// TwinCAT 3 PLC project ShutterMotion
// ProgramVersion: 3.1.4020.4
// libraries:
//   Tc2_Drive, * (Beckhoff Automation GmbH)
//   Tc2_EtherCAT, * (Beckhoff Automation GmbH)
//   Tc2_MC2, * (Beckhoff Automation GmbH)
//   Tc2_MC2_Drive, * (Beckhoff Automation GmbH)
//   Tc2_NcDrive, * (Beckhoff Automation GmbH)
//   Tc2_Standard, * (Beckhoff Automation GmbH)
//   Tc2_System, * (Beckhoff Automation GmbH)
//   Tc2_Utilities, * (Beckhoff Automation GmbH)
//   Tc3_MC2_AdvancedHoming, * (Beckhoff Automation GmbH)
//   Tc3_Module, * (Beckhoff Automation GmbH)
//   Util, * (System)
//   VisuDialogs, * (System)
// project tree:
//   DUTs/AxisStruct/ ST_AxisGroup.TcDUT, ST_Hall.TcDUT, ST_Track.TcDUT
//   DUTs/CCSInterface STRUCT/CCS to PLC/ ST_Calibrate.TcDUT, ST_ChangeAxisEnable.TcDUT, ST_ChangeBrakeState.TcDUT, ST_ClearAllFaults.TcDUT, ST_ClearAxisFaults.TcDUT, ST_CloseShutter.TcDUT, ST_DisableAllAxes.TcDUT, ST_EnableAllAxes.TcDUT, ST_GoToProd.TcDUT, ST_HomeAxis.TcDUT, ST_MoveAxisAbsolute.TcDUT, ST_MoveAxisRelative.TcDUT, ST_OpenShutter.TcDUT, ST_Reset.TcDUT, ST_TakeExposure.TcDUT, ST_ToggleSafetyCheck.TcDUT
//   DUTs/CCSInterface STRUCT/PLC to CCS/ AxisStatus.TcDUT, ST_CalibDone.TcDUT, ST_Disable.TcDUT, ST_Enable.TcDUT, ST_EncoderSample.TcDUT, ST_Error.TcDUT, ST_HallTransition.TcDUT, ST_Ignored.TcDUT, ST_MotionDone.TcDUT, ST_ShutterStatus.TcDUT, ST_Timer.TcDUT
//   DUTs/CCSInterface STRUCT/ ST_MsgToCCS.TcDUT, ST_MsgToPLC.TcDUT, ST_PLCMsg.TcDUT
//   DUTs/ENUM/ E_Commands.TcDUT, E_Components.TcDUT
//   DUTs/ENUM/State ENUM/ E_StatesEnabled.TcDUT, E_StatesMaint.TcDUT, E_StatesProd.TcDUT, E_StatesTop.TcDUT
//   DUTs/ ST_PtpDiag.TcDUT, T_MioSysTimes.TcDUT, T_TaskStartTimes.TcDUT
//   / GlobalTextList.TcGTLO, PlcTaskMain.TcTTO, Visualization Manager.TcVMO (not stored)
//   GVLs/ GVL.TcGVL
//   POUs/ FB_Power.TcPOU, FB_Protection.TcPOU, FB_PtpDiagReader.TcPOU, F_MioExtTime.TcPOU, F_HaveDifferentIDs.TcPOU, MAIN.TcPOU
//   POUs/StateMachine/ FB_Cycler.TcPOU, FB_ShutterSM.TcPOU, FB_Tracking.TcPOU
//   POUs/StateMachine/StateTop/ FB_StateDisabled.TcPOU, FB_StateEnabled.TcPOU
//   POUs/StateMachine/StateTop/StateEnabled/ FB_Reset.TcPOU, FB_StateMaint.TcPOU, FB_StateProd.TcPOU
//   POUs/StateMachine/StateTop/StateEnabled/StateMaint/ FB_Homing.TcPOU, FB_StateCalibrating.TcPOU, FB_StateMoving.TcPOU, FB_StateStill.TcPOU
//   POUs/StateMachine/StateTop/StateEnabled/StateProd/ FB_StateClosed.TcPOU, FB_StateClosing.TcPOU, FB_StateOpened.TcPOU, FB_StateOpening.TcPOU, FB_StateTravelling.TcPOU
//   VISUs/ Visualization.TcVIS
// real-time tasks:
//   TASK PlcTaskMain: cycle T#500us, priority 20, ADS port 350
// motion (NC):
//   TASK NC-Task 1 SAF: cycle T#500us, priority 1, ADS port 501
//   TASK NC-Task 1 SVB: cycle T#5ms, priority 40, ADS port 511
//   AXIS XP (id 1)
//     Dynamic: Acceleration=7407.41, Deceleration=7407.41, Jerk=32921.8
//     Velo: RefSearch=60, SlowManual=150
//     OtherSettings: AllowMotionCmdToSlave=true
//     encoder EncType=4
//       EncPara: ScaleFactorNumerator=0.0498327596, MaxCount=#x0000ffff
//         SoftEndMaxControl: Range=749
//         Inc: RefSearchInverse=true, RefSyncInverse=false, RefSoftSyncMask=#x0000ffff
//         TimeComp: TimeCompMode=1, EncDelayCycles=4
//     drive DrvType=24
//       Analog: VeloReferenz=2038.894
//       TimeComp: TaskDelayCycles=1
//     controller CtrType=1
//       CtrPara: PriorControlFactor=1
//         PosDiffControl: Range=2.5, Time=0.01
//         Observer: BandWidth=20
//   AXIS XM (id 2)
//     Dynamic: Acceleration=7407.41, Deceleration=7407.41, Jerk=32921.8
//     Velo: RefSearch=60
//     OtherSettings: AllowMotionCmdToSlave=true
//     encoder EncType=4
//       EncPara: ScaleFactorNumerator=0.0498327596, MaxCount=#x0000ffff
//         SoftEndMaxControl: Range=749
//         Inc: RefSoftSyncMask=#x0000ffff
//         TimeComp: TimeCompMode=1, EncDelayCycles=4
//     drive DrvType=24
//       Analog: VeloReferenz=2038.894
//       TimeComp: TaskDelayCycles=1
//     controller CtrType=1
//       CtrPara: PriorControlFactor=1
//         PosDiffControl: Range=2.5, Time=0.01
//         Observer: BandWidth=20
// I/O:
//   DEVICE Device 1 (EtherCAT), AmsNetId 10.0.1.28.2.1
//     MCD-00 (EK1200) [EK1200-5000 EtherCAT Power supply (2A E-Bus)]
//       MBC-00 (EL9570) [EL9570 Buffer capacitor terminal]
//       MDR-00 (EL7047) [EL7047 1Ch. Stepper motor output stage (50V, 5A)]
//       MPD-00 (EL9184) [EL9184 Potential Connection, 8 x 24V, 8 x Ground]
//       MIO-00 (EL1259) [EL1259 8Ch. Dig Input 24V/8Ch. Dig. Output 24V with Multi-Time-Stamp]
//       MIO-01 (EL1259) [EL1259 8Ch. Dig Input 24V/8Ch. Dig. Output 24V with Multi-Time-Stamp]
//       MTC-00 (EL3214) [EL3214 4Ch. Ana. Input PT100 (RTD)]
//       MBC-01 (EL9570) [EL9570 Buffer capacitor terminal]
//       MDR-01 (EL7047) [EL7047 1Ch. Stepper motor output stage (50V, 5A)]
//       MRE-01 (EL2622) [EL2622 2Ch. Relay Output, NO (230V AC / 30V DC)]
//       MTM-00 (EL6688) [EL6688 - External Synchronisation Interface (IEEE1588)]
//       END (EL9011) [EL9011 End Terminal]
// variable links:
//   (this object) <-> Device 1 (EtherCAT)/MCD-00 (EK1200)/MDR-00 (EL7047)
//     Drive/Inputs/In/nState1 @bit 3 <-> STM Status/Status/Error
//     Drive/Inputs/In/nState1 @bit 7 <-> STM Status/Status/Motor stall
//     Drive/Inputs/In/nState1 @bit 5 <-> STM Status/Status/Moving negative
//     Drive/Inputs/In/nState1 @bit 4 <-> STM Status/Status/Moving positive
//     Drive/Inputs/In/nState1 @bit 1 <-> STM Status/Status/Ready
//     Drive/Inputs/In/nState1 <-> STM Status/Status/Ready to enable
//     Drive/Inputs/In/nState1 @bit 6 <-> STM Status/Status/Torque reduced
//     Drive/Inputs/In/nState1 @bit 2 <-> STM Status/Status/Warning
//     Drive/Inputs/In/nState2 @bit 5 <-> STM Status/Status/Sync error
//     Drive/Inputs/In/nState2 @bit 7 <-> STM Status/Status/TxPDO Toggle
//     Drive/Inputs/In/nState4 @bit 1 <-> WcState/InputToggle
//     Drive/Outputs/Out/nCtrl1 <-> STM Control/Control/Enable
//     Drive/Outputs/Out/nCtrl1 @bit 2 <-> STM Control/Control/Reduce torque
//     Drive/Outputs/Out/nCtrl1 @bit 1 <-> STM Control/Control/Reset
//     Drive/Outputs/Out/nCtrl2 @bit 3 <-> STM Control/Control/Digital output 1
//     Drive/Outputs/Out/nDataOut2[0] <-> STM Velocity/Velocity
//     Enc/Inputs/In/nDataIn1[0] <-> ENC Status compact/Counter value
//     Enc/Inputs/In/nDataIn2[0] <-> ENC Status compact/Latch value
//     Enc/Inputs/In/nState1 @bit 4 <-> ENC Status compact/Status/Counter overflow
//     Enc/Inputs/In/nState1 @bit 3 <-> ENC Status compact/Status/Counter underflow
//     Enc/Inputs/In/nState1 @bit 7 <-> ENC Status compact/Status/Extrapolation stall
//     Enc/Inputs/In/nState1 <-> ENC Status compact/Status/Latch C valid
//     Enc/Inputs/In/nState1 @bit 1 <-> ENC Status compact/Status/Latch extern valid
//     Enc/Inputs/In/nState1 @bit 2 <-> ENC Status compact/Status/Set counter done
//     Enc/Inputs/In/nState2 @bit 4 <-> ENC Status compact/Status/Status of extern latch
//     Enc/Inputs/In/nState2 <-> ENC Status compact/Status/Status of input A
//     Enc/Inputs/In/nState2 @bit 1 <-> ENC Status compact/Status/Status of input B
//     Enc/Inputs/In/nState2 @bit 2 <-> ENC Status compact/Status/Status of input C
//     Enc/Inputs/In/nState2 @bit 5 <-> ENC Status compact/Status/Sync error
//     Enc/Inputs/In/nState2 @bit 7 <-> ENC Status compact/Status/TxPDO Toggle
//     Enc/Inputs/In/nState4 @bit 1 <-> WcState/InputToggle
//     Enc/Outputs/Out/nCtrl1 <-> ENC Control compact/Control/Enable latch C
//     Enc/Outputs/Out/nCtrl1 @bit 3 <-> ENC Control compact/Control/Enable latch extern on negative edge
//     Enc/Outputs/Out/nCtrl1 @bit 1 <-> ENC Control compact/Control/Enable latch extern on positive edge
//     Enc/Outputs/Out/nCtrl1 @bit 2 <-> ENC Control compact/Control/Set counter
//     Enc/Outputs/Out/nDataOut1[0] <-> ENC Control compact/Set counter value
//   (this object) <-> Device 1 (EtherCAT)/MCD-00 (EK1200)/MDR-01 (EL7047)
//     Drive/Inputs/In/nState1 @bit 3 <-> STM Status/Status/Error
//     Drive/Inputs/In/nState1 @bit 7 <-> STM Status/Status/Motor stall
//     Drive/Inputs/In/nState1 @bit 5 <-> STM Status/Status/Moving negative
//     Drive/Inputs/In/nState1 @bit 4 <-> STM Status/Status/Moving positive
//     Drive/Inputs/In/nState1 @bit 1 <-> STM Status/Status/Ready
//     Drive/Inputs/In/nState1 <-> STM Status/Status/Ready to enable
//     Drive/Inputs/In/nState1 @bit 6 <-> STM Status/Status/Torque reduced
//     Drive/Inputs/In/nState1 @bit 2 <-> STM Status/Status/Warning
//     Drive/Inputs/In/nState2 @bit 5 <-> STM Status/Status/Sync error
//     Drive/Inputs/In/nState2 @bit 7 <-> STM Status/Status/TxPDO Toggle
//     Drive/Inputs/In/nState4 @bit 1 <-> WcState/InputToggle
//     Drive/Outputs/Out/nCtrl1 <-> STM Control/Control/Enable
//     Drive/Outputs/Out/nCtrl1 @bit 2 <-> STM Control/Control/Reduce torque
//     Drive/Outputs/Out/nCtrl1 @bit 1 <-> STM Control/Control/Reset
//     Drive/Outputs/Out/nCtrl2 @bit 3 <-> STM Control/Control/Digital output 1
//     Drive/Outputs/Out/nDataOut2[0] <-> STM Velocity/Velocity
//     Enc/Inputs/In/nDataIn1[0] <-> ENC Status compact/Counter value
//     Enc/Inputs/In/nDataIn2[0] <-> ENC Status compact/Latch value
//     Enc/Inputs/In/nState1 @bit 4 <-> ENC Status compact/Status/Counter overflow
//     Enc/Inputs/In/nState1 @bit 3 <-> ENC Status compact/Status/Counter underflow
//     Enc/Inputs/In/nState1 @bit 7 <-> ENC Status compact/Status/Extrapolation stall
//     Enc/Inputs/In/nState1 <-> ENC Status compact/Status/Latch C valid
//     Enc/Inputs/In/nState1 @bit 1 <-> ENC Status compact/Status/Latch extern valid
//     Enc/Inputs/In/nState1 @bit 2 <-> ENC Status compact/Status/Set counter done
//     Enc/Inputs/In/nState2 @bit 4 <-> ENC Status compact/Status/Status of extern latch
//     Enc/Inputs/In/nState2 <-> ENC Status compact/Status/Status of input A
//     Enc/Inputs/In/nState2 @bit 1 <-> ENC Status compact/Status/Status of input B
//     Enc/Inputs/In/nState2 @bit 2 <-> ENC Status compact/Status/Status of input C
//     Enc/Inputs/In/nState2 @bit 5 <-> ENC Status compact/Status/Sync error
//     Enc/Inputs/In/nState2 @bit 7 <-> ENC Status compact/Status/TxPDO Toggle
//     Enc/Inputs/In/nState4 @bit 1 <-> WcState/InputToggle
//     Enc/Outputs/Out/nCtrl1 <-> ENC Control compact/Control/Enable latch C
//     Enc/Outputs/Out/nCtrl1 @bit 3 <-> ENC Control compact/Control/Enable latch extern on negative edge
//     Enc/Outputs/Out/nCtrl1 @bit 1 <-> ENC Control compact/Control/Enable latch extern on positive edge
//     Enc/Outputs/Out/nCtrl1 @bit 2 <-> ENC Control compact/Control/Set counter
//     Enc/Outputs/Out/nDataOut1[0] <-> ENC Control compact/Set counter value
//   ShutterMotion Instance <-> Device 1 (EtherCAT)
//     PlcTaskMain Inputs/GVL.DcToExtTimeOffset <-> InfoData/DcToExtTimeOffset
//     PlcTaskMain Inputs/GVL.DcToTcTimeOffset <-> InfoData/DcToTcTimeOffset
//   ShutterMotion Instance <-> Device 1 (EtherCAT)/MCD-00 (EK1200)/MDR-00 (EL7047)
//     PlcTaskMain Inputs/MAIN.fMotorTemp[0] <-> STM Synchron info data/Info data 1
//     PlcTaskMain Inputs/MAIN.stAxis[0].bLimitDeployed <-> STM Status/Status/Digital input 2
//     PlcTaskMain Inputs/MAIN.stAxis[0].bLimitHome <-> STM Status/Status/Digital input 1
//   ShutterMotion Instance <-> Device 1 (EtherCAT)/MCD-00 (EK1200)/MDR-01 (EL7047)
//     PlcTaskMain Inputs/MAIN.fMotorTemp[1] <-> STM Synchron info data/Info data 1
//     PlcTaskMain Inputs/MAIN.stAxis[1].bLimitDeployed <-> STM Status/Status/Digital input 2
//     PlcTaskMain Inputs/MAIN.stAxis[1].bLimitHome <-> STM Status/Status/Digital input 1
//   ShutterMotion Instance <-> Device 1 (EtherCAT)/MCD-00 (EK1200)/MIO-00 (EL1259)
//     PlcTaskMain Inputs/GVL.bInputEventState[{0..7}] <-> MTI Inputs 2x Channel {1..8}/Input event state 1  (8 links)
//     PlcTaskMain Inputs/GVL.mioSysTime[0] <-> DEV Inputs Device/SysTime
//     PlcTaskMain Inputs/GVL.nInputEventTime[{0..7}] <-> MTI Inputs 2x Channel {1..8}/Input event time 1  (8 links)
//     PlcTaskMain Inputs/GVL.nNumOfInputs[{0..7}] <-> MTI Inputs 2x Channel {1..8}/No of input events  (8 links)
//   ShutterMotion Instance <-> Device 1 (EtherCAT)/MCD-00 (EK1200)/MIO-01 (EL1259)
//     PlcTaskMain Inputs/GVL.bInputEventState[{8..14}] <-> MTI Inputs 2x Channel {1..7}/Input event state 1  (7 links)
//     PlcTaskMain Inputs/GVL.mioSysTime[1] <-> DEV Inputs Device/SysTime
//     PlcTaskMain Inputs/GVL.nInputEventTime[{8..14}] <-> MTI Inputs 2x Channel {1..7}/Input event time 1  (7 links)
//     PlcTaskMain Inputs/GVL.nNumOfInputs[{8..14}] <-> MTI Inputs 2x Channel {1..7}/No of input events  (7 links)
//   ShutterMotion Instance <-> Device 1 (EtherCAT)/MCD-00 (EK1200)/MRE-01 (EL2622)
//     PlcTaskMain Outputs/MAIN.stAxis[0].bBrake <-> Channel 1/Output
//     PlcTaskMain Outputs/MAIN.stAxis[1].bBrake <-> Channel 2/Output
//   ShutterMotion Instance <-> Device 1 (EtherCAT)/MCD-00 (EK1200)/MTC-00 (EL3214)
//     PlcTaskMain Inputs/MAIN.fRtdTemp[0] <-> RTD Inputs Channel 1/Value
//     PlcTaskMain Inputs/MAIN.fRtdTemp[1] <-> RTD Inputs Channel 2/Value
//     PlcTaskMain Inputs/MAIN.fRtdTemp[2] <-> RTD Inputs Channel 3/Value
//   ShutterMotion Instance <-> Device 1 (EtherCAT)/MCD-00 (EK1200)/MTM-00 (EL6688)
//     PlcTaskMain Inputs/GVL.ptpAdsAddr <-> InfoData/AdsAddr
//   ShutterMotion Instance <-> NC-Task 1 SAF/Axes/XM
//     PlcTaskMain Inputs/MAIN.stAxis[1].axisRef.NcToPlc <-> Outputs/ToPlc
//     PlcTaskMain Outputs/MAIN.stAxis[1].axisRef.PlcToNc <-> Inputs/FromPlc
//   ShutterMotion Instance <-> NC-Task 1 SAF/Axes/XP
//     PlcTaskMain Inputs/MAIN.stAxis[0].axisRef.NcToPlc <-> Outputs/ToPlc
//     PlcTaskMain Outputs/MAIN.stAxis[0].axisRef.PlcToNc <-> Inputs/FromPlc

CONFIGURATION ShutterMotion
    RESOURCE PLC ON TwinCAT3
        TASK PlcTaskMain(INTERVAL := T#500us, PRIORITY := 20);
        PROGRAM MAIN WITH PlcTaskMain : MAIN;
    END_RESOURCE
END_CONFIGURATION

// ---- DUTs/AxisStruct/ST_AxisGroup.TcDUT
TYPE ST_AxisGroup :
STRUCT
	//basic built in functions
	mcPower		: MC_Power;
	mcReset		: MC_Reset;
	mcMoveAbs	: MC_MoveAbsolute;
	mcMoveRel	: MC_MoveRelative;
	mcHome		: MC_Home;
	mcStop		: MC_Stop;
	mcJog		: MC_Jog; //required for homing routine
	
	//Status
	bIsCalibrated	: BOOL;
	
	//linkable variables
	axisRef					: AXIS_REF;;
	bBrake AT %Q* 			: BOOL;			(* 1-Brake disengaged, 0-Brake engaged *)
	bLimitHome AT %I*		: BOOL;			(* 1-at limit, 0-not at limit. Should be changed to 0-at limit, 1-not at limit to be SIL-2 compliance. Requires hardware change. *)
	bLimitDeployed AT %I*	: BOOL;			(* 1-at limit, 0-not at limit. Should be changed to 0-at limit, 1-not at limit to be SIL-2 compliance. Requires hardware change. *)

	//used for tracking linear motion using hall sensors
	//fbHallSig_rtrig		: ARRAY [GVL.cHallLower .. GVL.cHallUpper] OF R_TRIG;
	//fbHallSig_ftrig 	: ARRAY [GVL.cHallLower .. GVL.cHallUpper] OF F_TRIG;
	fHallPosCal			: ARRAY [GVL.cDirPos .. GVL.cDirNeg, 0 .. GVL.cTripCount] OF LREAL;
	fHallPosAct			: LREAL;
	nHallTime			: UDINT; //unit in nanosecond
	nTripCount 			: INT;
	//nHallSequence		: ARRAY [GVL.cDirPos .. GVL.cDirNeg, 0 .. GVL.cTripCount] OF WORD;
	stHall				: ARRAY [GVL.cDirPos .. GVL.cDirNeg, 0 .. GVL.cTripCount] OF ST_Hall;
	nSeqToCompare		: WORD;
	fPosDiffAtTrip		: LREAL;
	bTrackedFlag		: BOOL;

END_STRUCT
END_TYPE

// ---- DUTs/AxisStruct/ST_Hall.TcDUT
TYPE ST_Hall :
STRUCT
	nSeq	: WORD;
	bEdge	: BOOL; // 1-rising edge, 0-falling edge
END_STRUCT
END_TYPE

// ---- DUTs/AxisStruct/ST_Track.TcDUT
TYPE ST_Track :
STRUCT
	nSeqToCompare 	: WORD;
	bEdgeToCompare	: BOOL;
	tScanTime		: T_DCTIME64;
	nHallID			: DINT;
END_STRUCT
END_TYPE

// ---- DUTs/CCSInterface STRUCT/CCS to PLC/ST_Calibrate.TcDUT
{attribute 'pack_mode' := '1'}
TYPE ST_Calibrate EXTENDS ST_MsgToPLC:
STRUCT
    (* TBD - calibration parameters. *)
END_STRUCT
END_TYPE

// ---- DUTs/CCSInterface STRUCT/CCS to PLC/ST_ChangeAxisEnable.TcDUT
{attribute 'pack_mode' := '1'}
TYPE ST_ChangeAxisEnable EXTENDS ST_MsgToPLC:
STRUCT
    axisIndex	: DINT;
    enabled		: BOOL;
END_STRUCT
END_TYPE

// ---- DUTs/CCSInterface STRUCT/CCS to PLC/ST_ChangeBrakeState.TcDUT
{attribute 'pack_mode' := '1'}
TYPE ST_ChangeBrakeState EXTENDS ST_MsgToPLC:
STRUCT
	axisIndex	: DINT;
    state		: BOOL; (* TRUE=Disengaged, FALSE=Engaged *)
END_STRUCT
END_TYPE

// ---- DUTs/CCSInterface STRUCT/CCS to PLC/ST_ClearAllFaults.TcDUT
{attribute 'pack_mode' := '1'}
TYPE ST_ClearAllFaults EXTENDS ST_MsgToPLC:
STRUCT
END_STRUCT
END_TYPE

// ---- DUTs/CCSInterface STRUCT/CCS to PLC/ST_ClearAxisFaults.TcDUT
{attribute 'pack_mode' := '1'}
TYPE ST_ClearAxisFaults EXTENDS ST_MsgToPLC :
STRUCT
    axisIndex: DINT;
END_STRUCT
END_TYPE

// ---- DUTs/CCSInterface STRUCT/CCS to PLC/ST_CloseShutter.TcDUT
{attribute 'pack_mode' := '1'}
TYPE ST_CloseShutter EXTENDS ST_MsgToPLC:
STRUCT

END_STRUCT
END_TYPE

// ---- DUTs/CCSInterface STRUCT/CCS to PLC/ST_DisableAllAxes.TcDUT
{attribute 'pack_mode' := '1'}
TYPE ST_DisableAllAxes EXTENDS ST_MsgToPLC:
STRUCT
END_STRUCT
END_TYPE

// ---- DUTs/CCSInterface STRUCT/CCS to PLC/ST_EnableAllAxes.TcDUT
{attribute 'pack_mode' := '1'}
TYPE ST_EnableAllAxes EXTENDS ST_MsgToPLC:
STRUCT
END_STRUCT
END_TYPE

// ---- DUTs/CCSInterface STRUCT/CCS to PLC/ST_GoToProd.TcDUT
{attribute 'pack_mode' := '1'}
TYPE ST_GoToProd EXTENDS ST_MsgToPLC:
STRUCT
END_STRUCT
END_TYPE

// ---- DUTs/CCSInterface STRUCT/CCS to PLC/ST_HomeAxis.TcDUT
{attribute 'pack_mode' := '1'}
TYPE ST_HomeAxis EXTENDS ST_MsgToPLC:
STRUCT
    axisIndex: DINT;
END_STRUCT
END_TYPE

// ---- DUTs/CCSInterface STRUCT/CCS to PLC/ST_MoveAxisAbsolute.TcDUT
{attribute 'pack_mode' := '1'}
TYPE ST_MoveAxisAbsolute EXTENDS ST_MsgToPLC:
STRUCT
    axisIndex	: DINT;
    position	: LREAL;
    speed		: LREAL;
END_STRUCT
END_TYPE

// ---- DUTs/CCSInterface STRUCT/CCS to PLC/ST_MoveAxisRelative.TcDUT
{attribute 'pack_mode' := '1'}
TYPE ST_MoveAxisRelative EXTENDS ST_MsgToPLC:
STRUCT
    axisIndex	: DINT;
    distance	: LREAL;
    moveTime	: TIME;
END_STRUCT
END_TYPE

// ---- DUTs/CCSInterface STRUCT/CCS to PLC/ST_OpenShutter.TcDUT
{attribute 'pack_mode' := '1'}
TYPE ST_OpenShutter EXTENDS ST_MsgToPLC:
STRUCT

END_STRUCT
END_TYPE

// ---- DUTs/CCSInterface STRUCT/CCS to PLC/ST_Reset.TcDUT
{attribute 'pack_mode' := '1'}
TYPE ST_Reset EXTENDS ST_MsgToPLC:
STRUCT
    (* TBD - Shutter config info. *)
	speed 			: LREAL;
END_STRUCT
END_TYPE

// ---- DUTs/CCSInterface STRUCT/CCS to PLC/ST_TakeExposure.TcDUT
{attribute 'pack_mode' := '1'}
TYPE ST_TakeExposure EXTENDS ST_MsgToPLC:
STRUCT
    exposureTime: TIME;
END_STRUCT
END_TYPE

// ---- DUTs/CCSInterface STRUCT/CCS to PLC/ST_ToggleSafetyCheck.TcDUT
{attribute 'pack_mode' := '1'}
TYPE ST_ToggleSafetyCheck EXTENDS ST_MsgToPLC :
STRUCT
END_STRUCT
END_TYPE

// ---- DUTs/CCSInterface STRUCT/PLC to CCS/AxisStatus.TcDUT
{attribute 'pack_mode' := '1'}
(*already a built in struct called ST_AxisStatus so leaving this as AxisStatus instead*)
TYPE AxisStatus:
STRUCT
    actPos		: LREAL;	(* Actual position in mm. *)
    actVel		: LREAL;	(* Actual velocity in mm/sec. *)
    setAcc		: LREAL;	(* Set acceleration in mm/sec^2.*)
	enabled		: BOOL;		(* Is the axis enabled? *)
	brakeSet	: BOOL;		(* Is the brake engaged? *)
    lowLimit	: BOOL;		(* Low limit switch tripped? *)
	highLimit	: BOOL; 	(* High limit switch tripped? *)
	isHomed		: BOOL; 	(* Has the axis been homed? *)
	errorID		: UDINT; 	(* Axis error code. *)
    icTemp	: LREAL; 	    (* Temperature of motor controller IC, Celsius. *)
END_STRUCT
END_TYPE

// ---- DUTs/CCSInterface STRUCT/PLC to CCS/ST_CalibDone.TcDUT
{attribute 'pack_mode' := '1'}
TYPE ST_CalibDone EXTENDS ST_MsgToCCS:
STRUCT
    homePosition		: ARRAY [0..1] OF LREAL;
    deployedPosition	: ARRAY [0..1] OF LREAL;
    (* hallPosCal[a, d, t] is coordinate of
       the (t+1)st transition that occurred
       while moving axis a+1 in direction d.
       d=0 for positive, d=1 for negative.
     *)
    hallPosCal			: ARRAY [0..1, 0..1, 0..239] OF LREAL;
END_STRUCT
END_TYPE

// ---- DUTs/CCSInterface STRUCT/PLC to CCS/ST_Disable.TcDUT
{attribute 'pack_mode' := '1'}
TYPE ST_Disable EXTENDS ST_MsgToCCS:
STRUCT
END_STRUCT
END_TYPE

// ---- DUTs/CCSInterface STRUCT/PLC to CCS/ST_Enable.TcDUT
{attribute 'pack_mode' := '1'}
TYPE ST_Enable EXTENDS ST_MsgToCCS:
STRUCT
END_STRUCT
END_TYPE

// ---- DUTs/CCSInterface STRUCT/PLC to CCS/ST_EncoderSample.TcDUT
{attribute 'pack_mode' := '1'}
TYPE ST_EncoderSample:
STRUCT
    extTime	: T_DCTIME64; (* The time of the sample. Beckhoff TAI-like external time.*)
    pos		: LREAL; (* Axis position in mm. *)
END_STRUCT
END_TYPE

// ---- DUTs/CCSInterface STRUCT/PLC to CCS/ST_Error.TcDUT
{attribute 'pack_mode' := '1'}
TYPE ST_Error EXTENDS ST_MsgToCCS:
STRUCT
	errors	: UDINT;
END_STRUCT
END_TYPE

(*
TYPE E_Error:
(
    MOTION_VETOED 	:= 2#1,				//1,
    BRAKE_SET 		:= 2#10,			//2,
    HALL_DIFF 		:= 2#100,			//4,
    SHORT_EXPOSURE 	:= 2#1000,			//8,
    NOT_HOMED 		:= 2#10000,			//16,
    HOME_LIMIT 		:= 2#100000,		//32,
    DEPLOYED_LIMIT 	:= 2#1000000,		//64,
    UNSAFE_MOVE 	:= 2#10000000,		//128,
    TOO_FAST 		:= 2#100000000,		//256,
    AXIS_DISABLED 	:= 2#1000000000,	//512
) UDINT;
END_TYPE

*)

// ---- DUTs/CCSInterface STRUCT/PLC to CCS/ST_HallTransition.TcDUT
{attribute 'pack_mode' := '1'}
TYPE ST_HallTransition:
STRUCT
    id		: DINT; (* ID no. of sensor. *)
    extTime	: T_DCTIME64; (* The time of the transition, Beckhoff TAI-like external time. *)
    pos		: LREAL; (* Position of transition. *)
    on		: BOOL; (* TRUE for off -> on, else FALSE. *)
END_STRUCT
END_TYPE

// ---- DUTs/CCSInterface STRUCT/PLC to CCS/ST_Ignored.TcDUT
{attribute 'pack_mode' := '1'}
TYPE ST_Ignored EXTENDS ST_MsgToCCS:
STRUCT
    reason: DINT;
END_STRUCT
END_TYPE
 
(* Reasons for ignoring an event:
0: Wrong message-set version.
1: Wrong state.
*)

// ---- DUTs/CCSInterface STRUCT/PLC to CCS/ST_MotionDone.TcDUT
{attribute 'pack_mode' := '1'}
TYPE ST_MotionDone EXTENDS ST_MsgToCCS:
STRUCT
    axisNum		: DINT;						(* Which axis moved. *)
    startTime	: T_DCTIME64;				(* When motion started. Absolute TAI64N-like nanoseconds since Jan 1, 2000.*)
    startPos	: LREAL;					(* Starting position. *)
    targetDur	: LTIME;					(* Expected duration of motion. *)
    targetPos	: LREAL;					(* Desired final position. *)
    endPos		: LREAL;					(* Actual final position. *)
    actualDur	: LTIME;					(* Actual duration. *)
    ntrans		: DINT;						(* No. of Hall transitions. *)
    maxtrans	: DINT := GVL.cTripCount+1;	(* Size  N of trans array. *)
    nsamples	: DINT;						(* No of encoder samples. *)
    maxsamples	: DINT := GVL.cTripCount+1;	(* Size M of samples array. *)
    trans		: ARRAY [0 .. GVL.cTripCount] OF ST_HallTransition;
    samples		: ARRAY	[0 .. GVL.cTripCount] OF ST_EncoderSample;
	ptpState    : DINT;                     (* Encoded PTP slave clock state. *)
											(* 0=NO_OPERATION, 1=INITIALIZING, 2=FAULTY, 3=DISABLED, 4=LISTENING, *)
											(* 5=PRE_MASTER, 6=MASTER, 7=PASSIVE, 8=UNCALIBRATED, 9=SLAVE. *)
	leapSeconds : DINT;                     (* Latest leap second count gotten from PTP. *)
	leapIsValid : BOOL;                     (* Is nonzero if leap second count is valid, else is zero. *)
END_STRUCT
END_TYPE

// ---- DUTs/CCSInterface STRUCT/PLC to CCS/ST_ShutterStatus.TcDUT
{attribute 'pack_mode' := '1'}
TYPE ST_ShutterStatus EXTENDS ST_MsgToCCS:
STRUCT
    motionProfile	: DINT; (* Motion profile index. *)
    isCalibrated	: BOOL;
    smState			: DINT;
    axis			: ARRAY [0..1] OF AxisStatus;
	isSafetyOn		: BOOL;
	temperature 	: ARRAY [0..2] OF DINT;
	when			: T_DCTIME64;               (* When this message was created, TAI nanoseconds since Jan 1, 2000. *)
	ptpState    	: DINT;                     (* Encoded PTP slave clock state. *)
												(* 0=NO_OPERATION, 1=INITIALIZING, 2=FAULTY, 3=DISABLED, 4=LISTENING, *)
												(* 5=PRE_MASTER, 6=MASTER, 7=PASSIVE, 8=UNCALIBRATED, 9=SLAVE. *)
	leapSeconds		: DINT;                     (* Latest leap second count gotten from PTP. *)
	leapIsValid 	: BOOL;                     (* Is nonzero if leap second count is valid, else is zero. *)
END_STRUCT
END_TYPE

// ---- DUTs/CCSInterface STRUCT/PLC to CCS/ST_Timer.TcDUT
{attribute 'pack_mode' := '1'}
TYPE ST_Timer EXTENDS ST_MsgToCCS:
STRUCT
END_STRUCT
END_TYPE

// ---- DUTs/CCSInterface STRUCT/ST_MsgToCCS.TcDUT
{attribute 'pack_mode' := '1'}
TYPE ST_MsgToCCS EXTENDS ST_PLCMsg:
STRUCT
	sequence: DINT;(* Increment this to ensure notification. *)
END_STRUCT
END_TYPE

// ---- DUTs/CCSInterface STRUCT/ST_MsgToPLC.TcDUT
{attribute 'pack_mode' := '1'}
TYPE ST_MsgToPLC EXTENDS ST_PLCMsg:
STRUCT
    lowUUID		: LINT;	(* The low-order part of the UUID. *)
    highUUID	: LINT;	(* The high-order part of the UUID. *)
    dtime		: DINT;	(* Time of day of sending, in milliseconds. *)
    sequence	: DINT := 1;	(* Message sequence number. *)
END_STRUCT
END_TYPE

// ---- DUTs/CCSInterface STRUCT/ST_PLCMsg.TcDUT
{attribute 'pack_mode' := '1'}
TYPE ST_PLCMsg:
STRUCT
    version: DINT := GVL.nVersion; (* Version of set of PLC<->CCS messages. *)
END_STRUCT
END_TYPE

// ---- DUTs/ENUM/E_Commands.TcDUT
{attribute 'qualified_only'}
{attribute 'strict'}
TYPE E_Commands :
(
	noCommand,
	
	//Maint
	calibrate,
	changeAxisEnable,
	changeBrakeState,
	clearAllFaults,
	clearAxisFaults,
	disableAllAxes,
	enableAllAxes,
	goToProd,
	homeAxis,
	moveAxisAbsolute,
	moveAxisRelative,
	turnSafetyOff,
	
	//Prod
	openShutter,
	closeShutter,
	takeExposure,
	
	//Other
	reset
);
END_TYPE

// ---- DUTs/ENUM/E_Components.TcDUT
{attribute 'qualified_only'}
//{attribute 'strict'}
TYPE E_Components :
(
	motorXP,
	motorXM,
	brakes,
	terminals,
	controller,
	(*Leave 'system' as the last item on this list. 
	Any new components should be added before 'system' on this enum list, lest you break the code. *)
	system 
);
END_TYPE

// ---- DUTs/ENUM/State ENUM/E_StatesEnabled.TcDUT
{attribute 'qualified_only'}
{attribute 'strict'}
TYPE E_StatesEnabled :
(
	Maint 	:=	21000,
	Prod 	:=	22000 
) DINT;
END_TYPE

// ---- DUTs/ENUM/State ENUM/E_StatesMaint.TcDUT
{attribute 'qualified_only'}
{attribute 'strict'}
TYPE E_StatesMaint :
(
	Still 		:=	21010,
	Calibrating	:=	21020,
	Moving		:=	21030
) DINT;
END_TYPE

// ---- DUTs/ENUM/State ENUM/E_StatesProd.TcDUT
{attribute 'qualified_only'}
{attribute 'strict'}
TYPE E_StatesProd :
(
	Closed		:=	22040,
	Opening		:=	22050,
	Opened		:= 	22060,
	Closing		:= 	22070,
	Traveling	:=	22080
) DINT;
END_TYPE

// ---- DUTs/ENUM/State ENUM/E_StatesTop.TcDUT
{attribute 'qualified_only'}
{attribute 'strict'}
TYPE E_StatesTop :
(
	Disabled	:=	10000,
	Enabled		:=	20000
) DINT;
END_TYPE

// ---- DUTs/ST_PtpDiag.TcDUT
{attribute 'pack_mode' := '1'}
TYPE ST_PtpDiag : // Holds the data from the PTP Diag section of the EL6688 CoE items
STRUCT
	numMembers: UINT;  // Added by FB_EcCoESdoReadEx.
	PTPVersion: UINT;
	PTPState: UINT;
	ClockIdentity: ARRAY[0..7] OF BYTE;
	ParentPortIdentity: ARRAY[0..9] OF BYTE;
	GramdmasterIdentity: ARRAY [0..7] OF BYTE;
	OffsetFromMaster: DINT;
	MeanPathDelay:UDINT;
	StepsRemoved: UINT;
	SyncSequece: UINT;
	Timescale: UINT;
	CurrentUtcOffset: INT;
	CurrentUtcOffsetIsValid: UINT;
	Leap61: UINT;
	Leap59: UINT;
	EpochNumber: UINT;
END_STRUCT
END_TYPE

// ---- DUTs/T_MioSysTimes.TcDUT
TYPE T_MioSysTimes : ARRAY [0 .. GVL.cTimeBufferDepth] OF ARRAY [GVL.cMio0 .. GVL.cMio1] OF ULINT; END_TYPE

// ---- DUTs/T_TaskStartTimes.TcDUT
TYPE T_TaskStartTimes : ARRAY[0 .. GVL.cTimeBufferDepth] OF T_DCTIME64; END_TYPE

// ---- GVLs/GVL.TcGVL
{attribute 'qualified_only'}
VAR_GLOBAL CONSTANT
	
(*
			============================GENERAL SHUTTER LAYOUT===============================
			  ________________________________________________________________________________
	        ||                                  HALL SWITCH                                   \
	X- side ||       ----14---13--12---11---10---9---8---7---6---5---4---3---2--1---0----      \    X+ side
			||_________________________________________________________________________         \	
			| | 				 |                 **  **  **                 |        \ MotorXP \
			| |					 |            *                  *            |         \ MotorXM \   
			| |					 |         *                        *         |          \_________\
			| |				     |       *                            *       |                   | |
			| |					 |      *                              *      |                   | |
			| |		     	     |     *                                *     |                   | |
			| |		BLADE 	     |     *            APERTURE            *     |       BLADE       | |
			| |		STACK	     |     *                                *     |       STACK       | |
			| |		 XM 	     |     *                                *     |        XP         | |
			| |					 |      *                              *      |                   | |
			| |					 |       *                            *       |                   | |
			| |					 |         *                        *         |                   | |
			| |					 |   	      *                  *            |                   | |
			|_|__________________|_________________**  **  **_________________|___________________|_|
			
			       ---Negative-Direction--->                          <---Positive-Direction---
*)

	 
	cHallLower 		: INT := 0;
	cHallUpper 		: INT := 14;
	cDirPos			: INT := 0;
	cDirNeg			: INT := 1;
	cTripPerHall	: INT := 16;
	cNumOfHall		: INT := 15;
	cTripCount		: INT := (cTripPerHall*cNumOfHall)-1;
	cMio0           : INT := 0;  // Identifies the first multi-timestamping digital I/O module, MIO-00.
	cMio1           : INT := 1;  // Identifies the second MIO module, MIO-01.
	cFirstMio1Hall  : INT := 8;  // Hall sensors with this ID or greater are on the second MIO, MIO-01.
	  
	cBrakeOff		: BOOL	:= TRUE;
	cBrakeOn		: BOOL	:= FALSE;
	cScanVel		: LREAL := 30;//60;
	cHomeVel		: LREAL	:= 1;
	cCalibrateVel	: LREAL	:= 100;
	cPositionVel	: LREAL := 300;
	cPosStart		: LREAL := 0;
	cPosEnd			: LREAL := 750.76; //this will need to change for production once keyance snesors are in
	
	//For indexing axis
	cXP : INT := 0;  // +X side.
	cXM : INT := 1;  // -X side.
	
	// For how many cycles should we save PLC external task-start time and MIO SysTimes?
	cTimeBufferDepth: INT := 5;
	
	// Version number for the set of messages passsing between CCS and this firmware.
	nVersion		: DINT := 3;
	
END_VAR
VAR_GLOBAL
	//Safety State
	bSafetyOn	: BOOL := TRUE;
	
	//Hall Switches
	nHallSequence 			: WORD;
		
	// We're using our MIOs in synchronous multi-timestamping mode with a Multi-TimeStamping Factor (MTSF) of 2x. We expect at most one Hall event
	// per channel per cycle, so we've set the MTSF to 2x as recommended by the EL12xx manual.
	
	// SysTime is a 64-bit variable that in multi-timestamp mode contains the lower 32 bits of the MIO's DC clock. Each MIO channel reacts to a state change
	// by generating a timestamp that's a copy of the lower 32 bits of the current SysTime.
	
	{attribute 'TcLinkTo' := '[0] := TIID^Device 1 (EtherCAT)^MCD-00 (EK1200)^MIO-00 (EL1259)^DEV Inputs Device^SysTime;
	                          [1] := TIID^Device 1 (EtherCAT)^MCD-00 (EK1200)^MIO-01 (EL1259)^DEV Inputs Device^SysTime'}
	mioSysTime AT %I*: ARRAY [GVL.cMio0 .. GVL.cMio1] OF ULINT;  

	// The first event timestamp for each MIO channel that we use.
	{attribute 'TcLinkTo' := '
     [0]  := TIID^Device 1 (EtherCAT)^MCD-00 (EK1200)^MIO-00 (EL1259)^MTI Inputs 2x Channel 1^Input event time 1;
	 [1]  := TIID^Device 1 (EtherCAT)^MCD-00 (EK1200)^MIO-00 (EL1259)^MTI Inputs 2x Channel 2^Input event time 1;
	 [2]  := TIID^Device 1 (EtherCAT)^MCD-00 (EK1200)^MIO-00 (EL1259)^MTI Inputs 2x Channel 3^Input event time 1;
	 [3]  := TIID^Device 1 (EtherCAT)^MCD-00 (EK1200)^MIO-00 (EL1259)^MTI Inputs 2x Channel 4^Input event time 1;
	 [4]  := TIID^Device 1 (EtherCAT)^MCD-00 (EK1200)^MIO-00 (EL1259)^MTI Inputs 2x Channel 5^Input event time 1;
	 [5]  := TIID^Device 1 (EtherCAT)^MCD-00 (EK1200)^MIO-00 (EL1259)^MTI Inputs 2x Channel 6^Input event time 1;
	 [6]  := TIID^Device 1 (EtherCAT)^MCD-00 (EK1200)^MIO-00 (EL1259)^MTI Inputs 2x Channel 7^Input event time 1;
	 [7]  := TIID^Device 1 (EtherCAT)^MCD-00 (EK1200)^MIO-00 (EL1259)^MTI Inputs 2x Channel 8^Input event time 1;
	 [8]  := TIID^Device 1 (EtherCAT)^MCD-00 (EK1200)^MIO-01 (EL1259)^MTI Inputs 2x Channel 1^Input event time 1;
	 [9]  := TIID^Device 1 (EtherCAT)^MCD-00 (EK1200)^MIO-01 (EL1259)^MTI Inputs 2x Channel 2^Input event time 1;
	 [10] := TIID^Device 1 (EtherCAT)^MCD-00 (EK1200)^MIO-01 (EL1259)^MTI Inputs 2x Channel 3^Input event time 1;
	 [11] := TIID^Device 1 (EtherCAT)^MCD-00 (EK1200)^MIO-01 (EL1259)^MTI Inputs 2x Channel 4^Input event time 1;
	 [12] := TIID^Device 1 (EtherCAT)^MCD-00 (EK1200)^MIO-01 (EL1259)^MTI Inputs 2x Channel 5^Input event time 1;
	 [13] := TIID^Device 1 (EtherCAT)^MCD-00 (EK1200)^MIO-01 (EL1259)^MTI Inputs 2x Channel 6^Input event time 1;
	 [14] := TIID^Device 1 (EtherCAT)^MCD-00 (EK1200)^MIO-01 (EL1259)^MTI Inputs 2x Channel 7^Input event time 1'}
	nInputEventTime	AT %I*	: ARRAY [cHallLower .. cHallUpper] OF UDINT;

	// The input event count for each MIO channel that we use.
	{attribute 'TcLinkTo' := '
     [0]  := TIID^Device 1 (EtherCAT)^MCD-00 (EK1200)^MIO-00 (EL1259)^MTI Inputs 2x Channel 1^No of input events;
	 [1]  := TIID^Device 1 (EtherCAT)^MCD-00 (EK1200)^MIO-00 (EL1259)^MTI Inputs 2x Channel 2^No of input events;
	 [2]  := TIID^Device 1 (EtherCAT)^MCD-00 (EK1200)^MIO-00 (EL1259)^MTI Inputs 2x Channel 3^No of input events;
	 [3]  := TIID^Device 1 (EtherCAT)^MCD-00 (EK1200)^MIO-00 (EL1259)^MTI Inputs 2x Channel 4^No of input events;
	 [4]  := TIID^Device 1 (EtherCAT)^MCD-00 (EK1200)^MIO-00 (EL1259)^MTI Inputs 2x Channel 5^No of input events;
	 [5]  := TIID^Device 1 (EtherCAT)^MCD-00 (EK1200)^MIO-00 (EL1259)^MTI Inputs 2x Channel 6^No of input events;
	 [6]  := TIID^Device 1 (EtherCAT)^MCD-00 (EK1200)^MIO-00 (EL1259)^MTI Inputs 2x Channel 7^No of input events;
	 [7]  := TIID^Device 1 (EtherCAT)^MCD-00 (EK1200)^MIO-00 (EL1259)^MTI Inputs 2x Channel 8^No of input events;
	 [8]  := TIID^Device 1 (EtherCAT)^MCD-00 (EK1200)^MIO-01 (EL1259)^MTI Inputs 2x Channel 1^No of input events;
	 [9]  := TIID^Device 1 (EtherCAT)^MCD-00 (EK1200)^MIO-01 (EL1259)^MTI Inputs 2x Channel 2^No of input events;
	 [10] := TIID^Device 1 (EtherCAT)^MCD-00 (EK1200)^MIO-01 (EL1259)^MTI Inputs 2x Channel 3^No of input events;
	 [11] := TIID^Device 1 (EtherCAT)^MCD-00 (EK1200)^MIO-01 (EL1259)^MTI Inputs 2x Channel 4^No of input events;
	 [12] := TIID^Device 1 (EtherCAT)^MCD-00 (EK1200)^MIO-01 (EL1259)^MTI Inputs 2x Channel 5^No of input events;
	 [13] := TIID^Device 1 (EtherCAT)^MCD-00 (EK1200)^MIO-01 (EL1259)^MTI Inputs 2x Channel 6^No of input events;
	 [14] := TIID^Device 1 (EtherCAT)^MCD-00 (EK1200)^MIO-01 (EL1259)^MTI Inputs 2x Channel 7^No of input events'}
	nNumOfInputs AT %I*		: ARRAY [cHallLower .. cHallUpper] OF USINT;

	// Indicates for each channel whether the event was caused by a rising (1) or a falling (0) edge.
	{attribute 'TcLinkTo' := '
    [0]  := TIID^Device 1 (EtherCAT)^MCD-00 (EK1200)^MIO-00 (EL1259)^MTI Inputs 2x Channel 1^Input event state 1;
	[1]  := TIID^Device 1 (EtherCAT)^MCD-00 (EK1200)^MIO-00 (EL1259)^MTI Inputs 2x Channel 2^Input event state 1;
	[2]  := TIID^Device 1 (EtherCAT)^MCD-00 (EK1200)^MIO-00 (EL1259)^MTI Inputs 2x Channel 3^Input event state 1;
	[3]  := TIID^Device 1 (EtherCAT)^MCD-00 (EK1200)^MIO-00 (EL1259)^MTI Inputs 2x Channel 4^Input event state 1;
	[4]  := TIID^Device 1 (EtherCAT)^MCD-00 (EK1200)^MIO-00 (EL1259)^MTI Inputs 2x Channel 5^Input event state 1;
	[5]  := TIID^Device 1 (EtherCAT)^MCD-00 (EK1200)^MIO-00 (EL1259)^MTI Inputs 2x Channel 6^Input event state 1;
	[6]  := TIID^Device 1 (EtherCAT)^MCD-00 (EK1200)^MIO-00 (EL1259)^MTI Inputs 2x Channel 7^Input event state 1;
	[7]  := TIID^Device 1 (EtherCAT)^MCD-00 (EK1200)^MIO-00 (EL1259)^MTI Inputs 2x Channel 8^Input event state 1;
	[8]  := TIID^Device 1 (EtherCAT)^MCD-00 (EK1200)^MIO-01 (EL1259)^MTI Inputs 2x Channel 1^Input event state 1;
	[9]  := TIID^Device 1 (EtherCAT)^MCD-00 (EK1200)^MIO-01 (EL1259)^MTI Inputs 2x Channel 2^Input event state 1;
	[10] := TIID^Device 1 (EtherCAT)^MCD-00 (EK1200)^MIO-01 (EL1259)^MTI Inputs 2x Channel 3^Input event state 1;
	[11] := TIID^Device 1 (EtherCAT)^MCD-00 (EK1200)^MIO-01 (EL1259)^MTI Inputs 2x Channel 4^Input event state 1;
	[12] := TIID^Device 1 (EtherCAT)^MCD-00 (EK1200)^MIO-01 (EL1259)^MTI Inputs 2x Channel 5^Input event state 1;
	[13] := TIID^Device 1 (EtherCAT)^MCD-00 (EK1200)^MIO-01 (EL1259)^MTI Inputs 2x Channel 6^Input event state 1;
	[14] := TIID^Device 1 (EtherCAT)^MCD-00 (EK1200)^MIO-01 (EL1259)^MTI Inputs 2x Channel 7^Input event state 1'}
	bInputEventState AT %I*	: ARRAY [cHallLower .. cHallUpper] OF BOOL;

	//Timer
	fbWaitTimer	: TON;
	
	//TestVariable
	fbWritePersistentData	: WritePersistentData;
	
	// Process data from the EtherCAT master. The time offset types are given as ULINT instead of LINT because
	// that's how the corresponding arguments to F_GetCurExtTime64() are declared.
	{attribute 'TcLinkTo' :=  'TIID^Device 1 (EtherCAT)^InfoData^DcToExtTimeOffset'}
	DcToExtTimeOffset AT %I*: ULINT;

    {attribute 'TcLinkTo' :=  'TIID^Device 1 (EtherCAT)^InfoData^DcToTcTimeOffset'}
	DcToTcTimeOffset AT %I*: ULINT;
	
	// Process data from the EL6688 PTP module, MTM-00.
	{attribute 'TcLinkTo' := 'TIID^Device 1 (EtherCAT)^MCD-00 (EK1200)^MTM-00 (EL6688)^InfoData^AdsAddr'}
	ptpAdsAddr AT %I*: AMSADDR;       // Used to contact the module for CoE data.


END_VAR

VAR_GLOBAL PERSISTENT // For million cycle test
	strokeXP	: UDINT;
	strokeXM	: UDINT;
END_VAR

// ---- POUs/MAIN.TcPOU
PROGRAM MAIN
VAR
	ptpDiagReader: FB_PtpDiagReader;
	ptpDiagInfo: ST_PtpDiag;

	//Axis
	{attribute 'TcLinkTo' := '	[0].bLimitHome		:= TIID^Device 1 (EtherCAT)^MCD-00 (EK1200)^MDR-00 (EL7047)^STM Status^Status^Digital input 1;
								[0].bLimitDeployed	:= TIID^Device 1 (EtherCAT)^MCD-00 (EK1200)^MDR-00 (EL7047)^STM Status^Status^Digital input 2;
								[0].bBrake			:= TIID^Device 1 (EtherCAT)^MCD-00 (EK1200)^MRE-01 (EL2622)^Channel 1^Output;
								[1].bLimitHome		:= TIID^Device 1 (EtherCAT)^MCD-00 (EK1200)^MDR-01 (EL7047)^STM Status^Status^Digital input 1;
								[1].bLimitDeployed	:= TIID^Device 1 (EtherCAT)^MCD-00 (EK1200)^MDR-01 (EL7047)^STM Status^Status^Digital input 2;
								[1].bBrake			:= TIID^Device 1 (EtherCAT)^MCD-00 (EK1200)^MRE-01 (EL2622)^Channel 2^Output'}
	stAxis		: ARRAY [GVL.cXP .. GVL.cXM] OF ST_AxisGroup;
	
	//state machine function block
	fbShutterSM	: FB_ShutterSM;
	
	//external input
	{attribute 'TcLinkTo' := '	[0] := TIID^Device 1 (EtherCAT)^MCD-00 (EK1200)^MDR-00 (EL7047)^STM Synchron info data^Info data 1;
								[1] := TIID^Device 1 (EtherCAT)^MCD-00 (EK1200)^MDR-01 (EL7047)^STM Synchron info data^Info data 1'}
	fMotorTemp	AT %I*		: ARRAY [0..1] OF UINT;  //temp in 1 degree C per increment

	{attribute 'TcLinkTo' := '	[0] := TIID^Device 1 (EtherCAT)^MCD-00 (EK1200)^MTC-00 (EL3214)^RTD Inputs Channel 1^Value;
								[1] := TIID^Device 1 (EtherCAT)^MCD-00 (EK1200)^MTC-00 (EL3214)^RTD Inputs Channel 2^Value;
								[2] := TIID^Device 1 (EtherCAT)^MCD-00 (EK1200)^MTC-00 (EL3214)^RTD Inputs Channel 3^Value'}
	fRtdTemp	AT %I*		: ARRAY [0..2] OF INT;

	//other function block and var
	fbPower		: FB_Power;
	fbProtect	: FB_Protection;
	fSpeedRel	: LREAL;
	fbTracking	: FB_Tracking;

	//Timing test vars
	fbInputRtrig	: R_trig;
	fbInputFtrig	: F_trig;
	
	//
	eCommand		: E_Commands;
	
	//communication IN
	inCalibrate, 			ackCalibrate			: ST_Calibrate			;//:= (version:=nVersion);
	inChangeAxisEnable,		ackChangeAxisEnable		: ST_ChangeAxisEnable	;//:= (version:=nVersion);
	inChangeBrakeState,		ackChangeBrakeState		: ST_ChangeBrakeState	;//:= (version:=nVersion);
	inClearAllFaults,		ackClearAllFaults		: ST_ClearAllFaults		;//:= (version:=nVersion);
	inClearAxisFaults,		ackClearAxisFaults		: ST_ClearAxisFaults	;//:= (version:=nVersion);
	inCloseShutter,			ackCloseShutter			: ST_CloseShutter		;//:= (version:=nVersion);
	inDisableAllAxes,		ackDisableAllAxes		: ST_DisableAllAxes		;//:= (version:=nVersion);
	inEnableAllAxes,		ackEnableAllAxes		: ST_EnableAllAxes		;//:= (version:=nVersion);
	inGoToProd,				ackGoToProd				: ST_GoToProd			;//:= (version:=nVersion);
	inHomeAxis,				ackHomeAxis				: ST_HomeAxis			;//:= (version:=nVersion);
	inMoveAxisAbsolute,		ackMoveAxisAbsolute		: ST_MoveAxisAbsolute	;//:= (version:=nVersion);
	inMoveAxisRelative,		ackMoveAxisRelative		: ST_MoveAxisRelative	;//:= (version:=nVersion);
	inOpenShutter,			ackOpenShutter			: ST_OpenShutter		;//:= (version:=nVersion);
	inReset,				ackReset				: ST_Reset				;//:= (version:=nVersion);
	inTakeExposure,			ackTakeExposure			: ST_TakeExposure		;//:= (version:=nVersion);
	inToggleSafetyCheck,	ackToggleSafetyCheck	: ST_ToggleSafetyCheck	;//:= (version:=nVersion);
	
	//communication OUT
	fbOutTimer			: TON;
	bVersionSet			: BOOL;
	outCalibDone		: ST_CalibDone;
	outDisable			: ST_Disable;
	outEnable			: ST_Enable;
	outError			: ST_Error;
	outIgnored			: ST_Ignored;
	outMotionDone		: ST_MotionDone;
	outShutterStatus	: ST_ShutterStatus;
	outTimer			: ST_Timer;
	
	//edge detection
	stDisable_ftrig		: F_TRIG;
	stDisable_rtrig		: R_TRIG;
	stError_rtrig		: R_TRIG;
	stExpoTimer_rtrig	: R_TRIG;
	stCalibDone_rtrig	: R_TRIG;
	
END_VAR
VAR CONSTANT
	//Will change later once motionProfile and version are decided
	nMotionProfile		: DINT := 0;
	tUpdateTimer		: TIME := T#2S;
	cMaxSpeedSafetyOFF	: LREAL := 1;
END_VAR

(*
SN001 scaling factor
motor 1: 0.0498281
motor 2: 0.0498517
*)
(*
SN002 scaling factor
motor 1: 0.0498327596
motor 2: 0.0498327596
*)

// Read PTP Diag info from the EL6688 once a second. Initially it will take a cycle or so for the data to be collected, shouldn't be a problem. *)
ptpDiagReader();
ptpDiagInfo := ptpDiagReader.diagInfo;

(*update Axis_Ref status*)
stAxis[GVL.cXP].axisRef.ReadStatus();
stAxis[GVL.cXM].axisRef.ReadStatus();

////////////////////////////////////////////////////////////////////
//CCS to PLC
////////////////////////////////////////////////////////////////////
(* Check for new messages from CCS *)
ACT_CheckNewMessage();

////////////////////////////////////////////////////////////////////
(*shutter protection module*)
////////////////////////////////////////////////////////////////////
ACT_Protection();
	
////////////////////////////////////////////////////////////////////
//Shutter State Machine
////////////////////////////////////////////////////////////////////
ACT_StateMachine();
	
////////////////////////////////////////////////////////////////////
//PLC to CCS
////////////////////////////////////////////////////////////////////
(*Set version*)
//ACT_SetVersion();

//Shutter Status---------------------------------
ACT_ShutterStatus();

////////////////////////////////////////////////////////////////////
//Other (tracking, temperature, etc.)
////////////////////////////////////////////////////////////////////

(*track motion of both blades*)
fbTracking(
	stAxis				:= stAxis, 
	eCommand			:= eCommand, 
	bMotionDone			:= fbShutterSM.bMotionDone, 
	inReset				:= inReset,
	inMoveAxisAbsolute	:= inMoveAxisAbsolute,
	inMoveAxisRelative	:= inMoveAxisRelative,
	stOutMotionDone		=> outMotionDone);

ACTION ACT_CheckNewMessage:
(* Check for new messages from CCS *)
eCommand := E_Commands.noCommand;
IF F_HaveDifferentIDs(inCalibrate, ackCalibrate) THEN
	ackCalibrate := inCalibrate;
	IF ackCalibrate.version <> GVL.nVersion THEN
		outIgnored.reason := 0; (*wrong version*)
		outIgnored.sequence := outIgnored.sequence + 1;
	ELSIF fbShutterSM.nSMState<>E_StatesMaint.Still THEN//AND ((fbShutterSM.nSMState<>E_StatesProd.Closing) OR (fbShutterSM.nSMState<>E_StatesProd.Traveling)) THEN
		outIgnored.reason := 1; (*ignored by state machine*)
		outIgnored.sequence := outIgnored.sequence + 1;
	ELSE
		eCommand := E_Commands.calibrate;
	END_IF
	
ELSIF F_HaveDifferentIDs(inChangeAxisEnable, ackChangeAxisEnable) THEN
	ackChangeAxisEnable	:= inChangeAxisEnable;
	IF ackChangeAxisEnable.version <> GVL.nVersion THEN
		outIgnored.reason := 0; (*wrong version*)
		outIgnored.sequence := outIgnored.sequence + 1;
	ELSIF fbShutterSM.nSMState <> E_StatesMaint.Still THEN //AND ((fbShutterSM.nSMState<>E_StatesProd.Closing) OR (fbShutterSM.nSMState<>E_StatesProd.Traveling)) THEN
		outIgnored.reason := 1; (*ignored by state machine*)
		outIgnored.sequence := outIgnored.sequence + 1;
	ELSE
		eCommand := E_Commands.changeAxisEnable;
	END_IF
	
ELSIF F_HaveDifferentIDs(inChangeBrakeState, ackChangeBrakeState) THEN
	ackChangeBrakeState	:= inChangeBrakeState;
	IF ackChangeBrakeState.version <> GVL.nVersion THEN
		outIgnored.reason := 0; (*wrong version*)
		outIgnored.sequence := outIgnored.sequence + 1;
	ELSIF fbShutterSM.nSMState <> E_StatesMaint.Still THEN //AND ((fbShutterSM.nSMState<>E_StatesProd.Closing) OR (fbShutterSM.nSMState<>E_StatesProd.Traveling)) THEN
		outIgnored.reason := 1; (*ignored by state machine*)
		outIgnored.sequence := outIgnored.sequence + 1;
	ELSE
		eCommand := E_Commands.changeBrakeState;
	END_IF
	
ELSIF F_HaveDifferentIDs(inClearAllFaults, ackClearAllFaults) THEN
	ackClearAllFaults := inClearAllFaults;
	IF ackClearAllFaults.version <> GVL.nVersion THEN
		outIgnored.reason := 0; (*wrong version*)
		outIgnored.sequence := outIgnored.sequence + 1;
	ELSIF fbShutterSM.nSMState <> E_StatesMaint.Still THEN //AND ((fbShutterSM.nSMState<>E_StatesProd.Closing) OR (fbShutterSM.nSMState<>E_StatesProd.Traveling)) THEN
		outIgnored.reason := 1; (*ignored by state machine*)
		outIgnored.sequence := outIgnored.sequence + 1;
	ELSE
		eCommand := E_Commands.clearAllFaults;
	END_IF
	
ELSIF F_HaveDifferentIDs(inClearAxisFaults, ackClearAxisFaults) THEN
	ackClearAxisFaults 	:= inClearAxisFaults;
	IF ackClearAxisFaults.version <> GVL.nVersion THEN
		outIgnored.reason := 0; (*wrong version*)
		outIgnored.sequence := outIgnored.sequence + 1;
	ELSIF fbShutterSM.nSMState <> E_StatesMaint.Still THEN //AND ((fbShutterSM.nSMState<>E_StatesProd.Closing) OR (fbShutterSM.nSMState<>E_StatesProd.Traveling)) THEN
		outIgnored.reason := 1; (*ignored by state machine*)
		outIgnored.sequence := outIgnored.sequence + 1;
	ELSE
		eCommand := E_Commands.clearAxisFaults;
	END_IF
	
ELSIF F_HaveDifferentIDs(inCloseShutter, ackCloseShutter) THEN
	ackCloseShutter 	:= inCloseShutter;
	IF ackCloseShutter.version <> GVL.nVersion THEN
		outIgnored.reason := 0; (*wrong version*)
		outIgnored.sequence := outIgnored.sequence + 1;
	ELSIF fbShutterSM.nSMState <> E_StatesProd.Opened THEN //AND ((fbShutterSM.nSMState<>E_StatesProd.Closing) OR (fbShutterSM.nSMState<>E_StatesProd.Traveling)) THEN
		outIgnored.reason := 1; (*ignored by state machine*)
		outIgnored.sequence := outIgnored.sequence + 1;
	ELSE
		eCommand := E_Commands.closeShutter;
	END_IF
	
ELSIF F_HaveDifferentIDs(inDisableAllAxes, ackDisableAllAxes) THEN
	ackDisableAllAxes :=  inDisableAllAxes;
	IF ackDisableAllAxes.version <> GVL.nVersion THEN
		outIgnored.reason := 0; (*wrong version*)
		outIgnored.sequence := outIgnored.sequence + 1;
	ELSIF fbShutterSM.nSMState <> E_StatesMaint.Still THEN //AND ((fbShutterSM.nSMState<>E_StatesProd.Closing) OR (fbShutterSM.nSMState<>E_StatesProd.Traveling)) THEN
		outIgnored.reason := 1; (*ignored by state machine*)
		outIgnored.sequence := outIgnored.sequence + 1;
	ELSE
		eCommand := E_Commands.disableAllAxes;
	END_IF
	
ELSIF F_HaveDifferentIDs( inEnableAllAxes, ackEnableAllAxes) THEN
	ackEnableAllAxes :=  inEnableAllAxes;
	IF ackEnableAllAxes.version <> GVL.nVersion THEN
		outIgnored.reason := 0; (*wrong version*)
		outIgnored.sequence := outIgnored.sequence + 1;
	ELSIF fbShutterSM.nSMState <> E_StatesMaint.Still THEN //AND ((fbShutterSM.nSMState<>E_StatesProd.Closing) OR (fbShutterSM.nSMState<>E_StatesProd.Traveling)) THEN
		outIgnored.reason := 1; (*ignored by state machine*)
		outIgnored.sequence := outIgnored.sequence + 1;
	ELSE
		eCommand := E_Commands.enableAllAxes;
	END_IF
	
ELSIF F_HaveDifferentIDs( inGoToProd, ackGoToProd) THEN
	ackGoToProd :=  inGoToProd;
	IF ackGoToProd.version <> GVL.nVersion THEN
		outIgnored.reason := 0; (*wrong version*)
		outIgnored.sequence := outIgnored.sequence + 1;
	ELSIF fbShutterSM.nSMState <> E_StatesMaint.Still THEN //AND ((fbShutterSM.nSMState<>E_StatesProd.Closing) OR (fbShutterSM.nSMState<>E_StatesProd.Traveling)) THEN
		outIgnored.reason := 1; (*ignored by state machine*)
		outIgnored.sequence := outIgnored.sequence + 1;
	ELSE
		eCommand := E_Commands.goToProd; 
	END_IF	
	
ELSIF F_HaveDifferentIDs( inHomeAxis, ackHomeAxis) THEN
	ackHomeAxis :=  inHomeAxis;
	IF ackHomeAxis.version <> GVL.nVersion THEN
		outIgnored.reason := 0; (*wrong version*)
		outIgnored.sequence := outIgnored.sequence + 1;
	ELSIF fbShutterSM.nSMState <> E_StatesMaint.Still THEN //AND ((fbShutterSM.nSMState<>E_StatesProd.Closing) OR (fbShutterSM.nSMState<>E_StatesProd.Traveling)) THEN
		outIgnored.reason := 1; (*ignored by state machine*)
		outIgnored.sequence := outIgnored.sequence + 1;
	ELSE
		eCommand := E_Commands.homeAxis;
	END_IF
	
ELSIF F_HaveDifferentIDs( inMoveAxisAbsolute, ackMoveAxisAbsolute) THEN
	ackMoveAxisAbsolute :=  inMoveAxisAbsolute;	
	IF ackMoveAxisAbsolute.version <> GVL.nVersion THEN
		outIgnored.reason := 0; (*wrong version*)
		outIgnored.sequence := outIgnored.sequence + 1;
	ELSIF fbShutterSM.nSMState <> E_StatesMaint.Still THEN //AND ((fbShutterSM.nSMState<>E_StatesProd.Closing) OR (fbShutterSM.nSMState<>E_StatesProd.Traveling)) THEN
		outIgnored.reason := 1; (*ignored by state machine*)
		outIgnored.sequence := outIgnored.sequence + 1;
	ELSE
		eCommand := E_Commands.moveAxisAbsolute;
	END_IF
	
ELSIF F_HaveDifferentIDs( inMoveAxisRelative, ackMoveAxisRelative) THEN
	ackMoveAxisRelative := inMoveAxisRelative;	
	IF ackMoveAxisRelative.version <> GVL.nVersion THEN
		outIgnored.reason := 0; (*wrong version*)
		outIgnored.sequence := outIgnored.sequence + 1;
	ELSIF fbShutterSM.nSMState <> E_StatesMaint.Still THEN
		outIgnored.reason := 1; (*ignored by state machine*)
		outIgnored.sequence := outIgnored.sequence + 1;
	ELSE
		eCommand := E_Commands.moveAxisRelative;
	END_IF
	
ELSIF F_HaveDifferentIDs(inOpenShutter, ackOpenShutter) THEN
	ackOpenShutter := inOpenShutter;
	IF ackOpenShutter.version <> GVL.nVersion THEN
		outIgnored.reason := 0; (*wrong version*)
		outIgnored.sequence := outIgnored.sequence + 1;
	ELSIF fbShutterSM.nSMState <> E_StatesProd.Closed THEN
		outIgnored.reason := 1; (*ignored by state machine*)
		outIgnored.sequence := outIgnored.sequence + 1;
	ELSE
		eCommand := E_Commands.openShutter;
	END_IF
	
ELSIF F_HaveDifferentIDs(inReset, ackReset) THEN
	ackReset := inReset;	
	IF ackReset.version <> GVL.nVersion THEN
		outIgnored.reason := 0; (*wrong version*)
		outIgnored.sequence := outIgnored.sequence + 1;
	ELSE
		eCommand := E_Commands.reset;
	END_IF
	
ELSIF F_HaveDifferentIDs(inTakeExposure, ackTakeExposure) THEN
	ackTakeExposure := inTakeExposure;	
	IF ackTakeExposure.version <> GVL.nVersion THEN
		outIgnored.reason := 0; (*wrong version*)
		outIgnored.sequence := outIgnored.sequence + 1;
	ELSIF fbShutterSM.nSMState <> E_StatesProd.Closed THEN
		outIgnored.reason := 1; (*ignored by state machine*)
		outIgnored.sequence := outIgnored.sequence + 1;
	ELSE
		eCommand := E_Commands.takeExposure;
	END_IF
	
ELSIF F_HaveDifferentIDs(inToggleSafetyCheck, ackToggleSafetyCheck) THEN
	ackToggleSafetyCheck := inToggleSafetyCheck;	
	IF ackToggleSafetyCheck.version <> GVL.nVersion THEN
		outIgnored.reason := 0; (*wrong version*)
		outIgnored.sequence := outIgnored.sequence + 1;
	ELSIF fbShutterSM.nSMState <> E_StatesMaint.Still THEN
		outIgnored.reason := 1; (*ignored by state machine*)
		outIgnored.sequence := outIgnored.sequence + 1;
	ELSE
		eCommand := E_Commands.turnSafetyOff;
	END_IF
	
END_IF
END_ACTION

ACTION ACT_Protection:
IF (eCommand = E_Commands.turnSafetyOff) THEN
	GVL.bSafetyOn := NOT GVL.bSafetyOn;
	outShutterStatus.sequence := outShutterStatus.sequence +1;
END_IF
IF (fbTracking.bMotionDone AND NOT GVL.bSafetyOn) THEN
	GVL.bSafetyOn := TRUE;
	outShutterStatus.sequence := outShutterStatus.sequence +1;
END_IF
outShutterStatus.isSafetyOn := GVL.bSafetyOn;

IF GVL.bSafetyOn THEN
	fbProtect(
		stAxis 				:= stAxis, 
		nState 				:= fbShutterSM.nSMState,
		eCommand 			:= eCommand,
		
		inCalibrate			:= inCalibrate,
		inChangeAxisEnable	:= inChangeAxisEnable,
		inChangeBrakeState	:= inChangeBrakeState,
		inClearAllFaults	:= inClearAllFaults,
		inClearAxisFaults	:= inClearAxisFaults,
		inCloseShutter		:= inCloseShutter,
		inDisableAllAxes	:= inDisableAllAxes,
		inEnableAllAxes		:= inEnableAllAxes,
		inGoToProd			:= inGoToProd,
		inHomeAxis			:= inHomeAxis,
		inMoveAxisAbsolute	:= inMoveAxisAbsolute,
		inMoveAxisRelative	:= inMoveAxisRelative,
		inOpenShutter		:= inOpenShutter,
		inReset				:= inReset,
		inTakeExposure		:= inTakeExposure,
		inToggleSafetyCheck	:= inToggleSafetyCheck);
ELSE
(* Shouldn't be able to enter PROD mode so this is not needed
	IF (inReset.speed > cMaxSpeedSafetyOFF) THEN
		inReset.speed := cMaxSpeedSafetyOFF;
	END_IF
*)	
	IF (inMoveAxisAbsolute.speed > cMaxSpeedSafetyOFF) THEN
		inMoveAxisAbsolute.speed := cMaxSpeedSafetyOFF;
	END_IF
	
	IF ((TIME_TO_LREAL(inMoveAxisRelative.moveTime)/1000)>0) THEN
		fSpeedRel	:= (2*ABS(inMoveAxisRelative.distance)/(TIME_TO_LREAL(inMoveAxisRelative.moveTime)/1000));
	ELSE
		fSpeedRel	:= 0.0001;
	END_IF
	
	if (fSpeedRel > cMaxSpeedSafetyOFF) THEN
		fSpeedRel := cMaxSpeedSafetyOFF;
		inMoveAxisRelative.moveTime := LREAL_TO_TIME(1000*2*ABS(inMoveAxisRelative.distance)/(fSpeedRel));
	END_IF
END_IF
END_ACTION

ACTION ACT_SetVersion:
(*Set version*)
IF NOT bVersionSet THEN
	bVersionSet 				:= TRUE;
	outShutterStatus.version 	:= GVL.nVersion;
	outDisable.version 			:= GVL.nVersion;
	outEnable.version 			:= GVL.nVersion;
	outError.version 			:= GVL.nVersion;
	outIgnored.version 			:= GVL.nVersion;
	outTimer.version 			:= GVL.nVersion;
	outCalibDone.version 		:= GVL.nVersion;
	outMotionDone.version		:= GVL.nVersion;
END_IF
END_ACTION

ACTION ACT_ShutterStatus:
//updates upon changes---------------------------------------------
//Shutter disabled/enabled
stDisable_rtrig(CLK:=(fbShutterSM.nSMState = E_StatesTop.Disabled));
IF stDisable_rtrig.Q THEN
	outDisable.sequence := outDisable.sequence + 1;
END_IF
stDisable_ftrig(CLK:=(fbShutterSM.nSMState = E_StatesTop.Disabled));
IF stDisable_ftrig.Q THEN
	outEnable.sequence := outEnable.sequence + 1;
END_IF

//Exposure timer ended
outTimer.sequence := fbShutterSM.stOutTimer.sequence;

//Calibration Done
stCalibDone_rtrig(CLK:=fbShutterSM.bCalibDone);
IF stCalibDone_rtrig.Q THEN
	outCalibDone.hallPosCal := fbShutterSM.stOutCalibDone.hallPosCal;
	outCalibDone.sequence := outCalibDone.sequence + 1;
	outShutterStatus.isCalibrated := (stAxis[GVL.cXP].bIsCalibrated AND stAxis[GVL.cXM].bIsCalibrated);
	outShutterStatus.sequence := outShutterStatus.sequence +1;
END_IF

//Periodic updates---------------------------------------------
fbOutTimer(IN:=TRUE, PT:=tUpdateTimer);
IF fbOutTimer.Q THEN
	fbOutTimer(IN:=FALSE);
	
	(*increment sequence*)
	outShutterStatus.sequence := outShutterStatus.sequence +1;

	(*shutter status update, common*)
	outShutterStatus.motionProfile := nMotionProfile;
	outShutterStatus.isCalibrated := (stAxis[GVL.cXP].bIsCalibrated AND stAxis[GVL.cXM].bIsCalibrated);
	outShutterStatus.smState := fbShutterSM.nSMState;
	outShutterStatus.temperature[0] := INT_TO_DINT(fRtdTemp[0]);
	outShutterStatus.temperature[1] := INT_TO_DINT(fRtdTemp[1]);
	outShutterStatus.temperature[2] := INT_TO_DINT(fRtdTemp[2]);
	outShutterStatus.when := F_GetCurExtTime64(GVL.DcToExtTimeOffset, GVL.DcToTcTimeOffset);
	outShutterStatus.ptpState := MAIN.ptpDiagInfo.PTPState;
	outShutterStatus.leapSeconds := MAIN.ptpDiagInfo.CurrentUtcOffset;
	outShutterStatus.leapIsValid := TO_BOOL(MAIN.ptpDiagInfo.CurrentUtcOffsetIsValid);
	
	(*shutter status update, axis XP specific*)
	outShutterStatus.axis[GVL.cXP].actPos := stAxis[GVL.cXP].axisRef.NcToPlc.ActPos;
	outShutterStatus.axis[GVL.cXP].actVel := stAxis[GVL.cXP].axisRef.NcToPlc.ActVelo;
	outShutterStatus.axis[GVL.cXP].setAcc := stAxis[GVL.cXP].axisRef.NcToPlc.SetAcc;
	outShutterStatus.axis[GVL.cXP].brakeSet := NOT stAxis[GVL.cXP].bBrake;
	outShutterStatus.axis[GVL.cXP].enabled := (stAxis[GVL.cXP].axisRef.PlcToNc.ControlDWord.0 AND	(*controlDword bit 0, 1, 2 corresponds to*)
												stAxis[GVL.cXP].axisRef.PlcToNc.ControlDWord.1 AND 	(*MC_Power parameters Enable, Enable_Positive, Enable_Negative*)
												stAxis[GVL.cXP].axisRef.PlcToNc.ControlDWord.2);
	outShutterStatus.axis[GVL.cXP].errorID	:= stAxis[GVL.cXP].axisRef.Status.ErrorID;
	outShutterStatus.axis[GVL.cXP].highLimit := stAxis[GVL.cXP].bLimitDeployed;
	outShutterStatus.axis[GVL.cXP].lowLimit := stAxis[GVL.cXP].bLimitHome;
	outShutterStatus.axis[GVL.cXP].isHomed := stAxis[GVL.cXP].axisRef.Status.Homed;
	outShutterStatus.axis[GVL.cXP].icTemp := UINT_TO_LREAL(fMotorTemp[0]);
	
	(*shutter status update, axis XM specific*)
	outShutterStatus.axis[GVL.cXM].actPos := stAxis[GVL.cXM].axisRef.NcToPlc.ActPos;
	outShutterStatus.axis[GVL.cXM].actVel := stAxis[GVL.cXM].axisRef.NcToPlc.ActVelo;
	outShutterStatus.axis[GVL.cXM].setAcc := stAxis[GVL.cXM].axisRef.NcToPlc.SetAcc;
	outShutterStatus.axis[GVL.cXM].brakeSet := NOT stAxis[GVL.cXM].bBrake;
	outShutterStatus.axis[GVL.cXM].enabled := (stAxis[GVL.cXM].axisRef.PlcToNc.ControlDWord.0 AND	(*controlDword bit 0, 1, 2 corresponds to*)
												stAxis[GVL.cXM].axisRef.PlcToNc.ControlDWord.1 AND 	(*MC_Power parameters Enable, Enable_Positive, Enable_Negative*)
												stAxis[GVL.cXM].axisRef.PlcToNc.ControlDWord.2);
	outShutterStatus.axis[GVL.cXM].errorID	:= stAxis[GVL.cXM].axisRef.Status.ErrorID;
	outShutterStatus.axis[GVL.cXM].highLimit := stAxis[GVL.cXM].bLimitHome;
	outShutterStatus.axis[GVL.cXM].lowLimit := stAxis[GVL.cXM].bLimitDeployed;
	outShutterStatus.axis[GVL.cXM].isHomed := stAxis[GVL.cXM].axisRef.Status.Homed;
	outShutterStatus.axis[GVL.cXM].icTemp := UINT_TO_LREAL(fMotorTemp[1]);
	
END_IF
END_ACTION

ACTION ACT_StateMachine:
fbShutterSM(
	//inputs
	stAxis				:= stAxis,
	eCommand			:= eCommand,
	stCalibrate			:= inCalibrate,
	stChangeAxisEnable	:= inChangeAxisEnable,
	stChangeBrakeState	:= inChangeBrakeState,
	stClearAllFaults	:= inClearAllFaults,
	stClearAxisFaults	:= inClearAxisFaults,
	stCloseShutter		:= inCloseShutter,
	stDisableAllAxes	:= inDisableAllAxes,
	stEnableAllAxes		:= inEnableAllAxes,
	stGoToProd			:= inGoToProd,
	stHomeAxis			:= inHomeAxis,
	stMoveAxisAbsolute	:= inMoveAxisAbsolute,
	stMoveAxisRelative	:= inMoveAxisRelative,
	stOpenShutter		:= inOpenShutter,
	stReset				:= inReset,
	stTakeExposure		:= inTakeExposure);
END_ACTION

END_PROGRAM

// ---- POUs/FB_PtpDiagReader.TcPOU
FUNCTION_BLOCK PUBLIC FB_PtpDiagReader
VAR_INPUT
END_VAR
VAR_OUTPUT
	diagInfo: ST_PtpDiag;
END_VAR
VAR
	running: BOOL := FALSE;
	first: BOOL := TRUE;
	netId: T_AmsNetId;
	port: UINT; 
	index: WORD := 16#FA80;
	subIndex: BYTE := 0;
	reader: FB_EcCoESdoReadEx;
	buf: ST_PtpDiag;
	readInterval: TIME := T#1S;
	timer: TON;
	c1: LINT := 0;
	c2: LINT := 0;
	c3: LINT := 0;
	c4: LINT := 0;
END_VAR

// The first time through, get the required ADS parameters.
IF first THEN
	first := FALSE;
	netId := F_CreateAmsNetId(GVL.ptpAdsAddr.netId);
	port := GVL.ptpAdsAddr.port;
	timer(IN:=TRUE, PT:=readInterval);
END_IF

timer();
// If a request is in progress then check for completion.
IF running THEN
	c1 := c1 + 1;
	reader(bExecute:=running);
	IF NOT reader.bBusy THEN
		c2 := c2 + 1;
		diagInfo := buf;
		running := FALSE;
		reader(bExecute:=running);
	END_IF
ELSE
	c3 := c3 + 1;
	IF timer.Q THEN
		timer(IN:=FALSE);
	    running := TRUE;
		timer(IN:=running);
	    reader(sNetId:=netId, nSlaveAddr:=port, nSubIndex:=subIndex, nIndex:=index, pDstBuf:=ADR(buf), cbBufLen:=SIZEOF(buf), bCompleteAccess:=TRUE, bExecute:=running);
	    IF reader.bBusy THEN
		    c4 := c4 + 1;
	    END_IF
	END_IF
END_IF

END_FUNCTION_BLOCK

// ---- POUs/StateMachine/FB_ShutterSM.TcPOU
FUNCTION_BLOCK FB_ShutterSM
VAR_IN_OUT
	stAxis  	: ARRAY [GVL.cXP .. GVL.cXM] OF ST_AxisGroup;
END_VAR
VAR_INPUT
	//commands
	eCommand			: E_Commands;
	stCalibrate			: ST_Calibrate;
	stChangeAxisEnable	: ST_ChangeAxisEnable;
	stChangeBrakeState	: ST_ChangeBrakeState;
	stClearAllFaults	: ST_ClearAllFaults;
	stClearAxisFaults	: ST_ClearAxisFaults;
	stCloseShutter		: ST_CloseShutter;
	stDisableAllAxes	: ST_DisableAllAxes;
	stEnableAllAxes		: ST_EnableAllAxes;
	stGoToProd			: ST_GoToProd;
	stHomeAxis			: ST_HomeAxis;
	stMoveAxisAbsolute	: ST_MoveAxisAbsolute;
	stMoveAxisRelative	: ST_MoveAxisRelative;
	stOpenShutter		: ST_OpenShutter;
	stReset				: ST_Reset;
	stTakeExposure		: ST_TakeExposure;
END_VAR
VAR_OUTPUT
	bCalibDone			: BOOL;
	bMotionDone			: BOOL;
	stOutCalibDone		: ST_CalibDone;
	stOutError			: ST_Error;
	stOutTimer			: ST_Timer;
	nSMState			: DINT;
END_VAR
VAR
	//state-machine
	eCurrentState	: E_StatesTop;
	eNextState		: E_StatesTop;
	fbEnabled		: FB_StateEnabled;
	fbDisabled		: FB_StateDisabled;
	bLowerEntry		: BOOL;

	//used in homeShutter Action
	fbHomeDelay : TON;

END_VAR

(* Top state of the shutter state machine *)
IF eCurrentState <> eNextState THEN
	bLowerEntry := TRUE;
END_IF

eNextState := E_StatesTop.Enabled;
eCurrentState := eNextState;
(*Start of state machine*)
CASE eCurrentState OF
	E_StatesTop.Disabled: 
		fbDisabled(
			stAxis 		:= stAxis, 
			btopEntry	:=bLowerEntry,
			nSMState	=> nSMState);

	E_StatesTop.Enabled:
		fbEnabled(
			//inputs
			stAxis 				:= stAxis, 
			bTopEntry 			:= bLowerEntry,
			eCommand			:= eCommand,
			stCalibrate			:= stCalibrate,
			stChangeAxisEnable	:= stChangeAxisEnable,
			stChangeBrakeState	:= stChangeBrakeState,
			stClearAllFaults	:= stClearAllFaults,
			stClearAxisFaults	:= stClearAxisFaults,
			stCloseShutter		:= stCloseShutter,
			stDisableAllAxes	:= stDisableAllAxes,
			stEnableAllAxes		:= stEnableAllAxes,
			stGoToProd			:= stGoToProd,
			stHomeAxis			:= stHomeAxis,
			stMoveAxisAbsolute	:= stMoveAxisAbsolute,
			stMoveAxisRelative	:= stMoveAxisRelative,
			stOpenShutter		:= stOpenShutter,
			stReset				:= stReset,
			stTakeExposure		:= stTakeExposure,
			//outputs
			bCalibDone			=> bCalibDone,
			bMotionDone			=> bMotionDone,
			stOutCalibDone		=> stOutCalibDone,
			stOutTimer			=> stOutTimer,
			nSMState			=> nSMState);
END_CASE

END_FUNCTION_BLOCK

// ---- POUs/StateMachine/StateTop/FB_StateEnabled.TcPOU
FUNCTION_BLOCK FB_StateEnabled
VAR_IN_OUT
	stAxis  	: ARRAY [GVL.cXP .. GVL.cXM] OF ST_AxisGroup;
	bTopEntry	: BOOL;
END_VAR
VAR_INPUT
	eCommand			: E_Commands;
	stCalibrate			: ST_Calibrate;
	stChangeAxisEnable	: ST_ChangeAxisEnable;
	stChangeBrakeState	: ST_ChangeBrakeState;
	stClearAllFaults	: ST_ClearAllFaults;
	stClearAxisFaults	: ST_ClearAxisFaults;
	stCloseShutter		: ST_CloseShutter;
	stDisableAllAxes	: ST_DisableAllAxes;
	stEnableAllAxes		: ST_EnableAllAxes;
	stGoToProd			: ST_GoToProd;
	stHomeAxis			: ST_HomeAxis;
	stMoveAxisAbsolute	: ST_MoveAxisAbsolute;
	stMoveAxisRelative	: ST_MoveAxisRelative;
	stOpenShutter		: ST_OpenShutter;
	stReset				: ST_Reset;
	stTakeExposure		: ST_TakeExposure;
END_VAR
VAR_OUTPUT
	bCalibDone			: BOOL;
	bMotionDone			: BOOL;
	stOutCalibDone		: ST_CalibDone;
	stOutTimer			: ST_Timer;
	nSMState			: DINT;
END_VAR
VAR
	//state-machine
	eCurrentState	: E_StatesEnabled;
	eNextState		: E_StatesEnabled;
	fbMaint			: FB_StateMaint;
	fbProd			: FB_StateProd;
	bLowerEntry		: BOOL;
	
	//Event
	bIsCalibrated	: BOOL;
	bShutterReady	: BOOL;

	//Other var
	fbReset			: FB_Reset;
	bResetting		: BOOL;
	bResetEntry		: BOOL;
	bStopping		: BOOL;
	
END_VAR

(**)
IF bTopEntry = TRUE THEN
	bTopEntry := FALSE;
	(*Check if shutter blade sets are calibrated. If not, then go to still, otherwise go to previous state*)
	IF stAxis[GVL.cXP].bIsCalibrated AND stAxis[GVL.cXM].bIsCalibrated THEN
		eNextState := eCurrentState;
	ELSE
		eNextState := E_StatesEnabled.Maint;
	END_IF
END_IF	

IF eCurrentState <> eNextState THEN
	bLowerEntry := TRUE;
END_IF
eCurrentState := eNextState;

(* State Machine *)
CASE eCurrentState OF
	
	E_StatesEnabled.Maint:
		fbMaint(
			//inputs
			stAxis 				:= stAxis, 
			bTopEntry 			:= bLowerEntry, 
			eCommand			:= eCommand,
			stCalibrate			:= stCalibrate,
			stChangeAxisEnable	:= stChangeAxisEnable,
			stChangeBrakeState	:= stChangeBrakeState,
			stClearAllFaults	:= stClearAllFaults,
			stClearAxisFaults	:= stClearAxisFaults,
			stDisableAllAxes	:= stDisableAllAxes,
			stEnableAllAxes		:= stEnableAllAxes,
			stGoToProd			:= stGoToProd,
			stHomeAxis			:= stHomeAxis,
			stMoveAxisAbsolute	:= stMoveAxisAbsolute,
			stMoveAxisRelative	:= stMoveAxisRelative,
			//outputs
			bCalibDone			=> bCalibDone,
			bMotionDone			=> bMotionDone,
			stOutCalibDone		=> stOutCalibDone,
			nSMState			=> nSMState);	
		IF bShutterReady AND eCommand = E_Commands.goToProd THEN
			eNextState := E_StatesEnabled.Prod;
		END_IF
	
	E_StatesEnabled.Prod:
		fbProd(
			//inputs
			stAxis			:= stAxis, 
			bTopEntry 		:= bLowerEntry,
			eCommand		:= eCommand,
			fSpeed			:= stReset.speed,
			stOpenShutter	:= stOpenShutter,
			stCloseShutter	:= stCloseShutter,
			stTakeExposure	:= stTakeExposure,
			//outputs
			bMotionDone		=> bMotionDone,
			nSMState		=> nSMState,
			stOutTimer		=> stOutTimer);

END_CASE

//Reset routine
IF eCommand = E_Commands.reset THEN
	bResetting 	:= TRUE;
	bResetEntry	:= TRUE;
END_IF
IF bResetting THEN
	fbReset(stAxis:=stAxis, bResetEntry:=bResetEntry,bResetting:=bResetting,);
	eNextState := E_StatesEnabled.Maint;
	bLowerEntry := TRUE; //forces states in Maint to go to still state
END_IF


//Status for when shutter is ready to be put into prod mode.
bShutterReady := (stAxis[GVL.cXP].bBrake AND stAxis[GVL.cXM].bBrake) AND (stAxis[GVL.cXP].bIsCalibrated AND stAxis[GVL.cXM].bIsCalibrated) AND
	(
		((stAxis[GVL.cXP].axisRef.NcToPlc.ActPos<1) AND (stAxis[GVL.cXM].axisRef.NcToPlc.ActPos<1)) OR 
		((stAxis[GVL.cXP].axisRef.NcToPlc.ActPos>750) AND (stAxis[GVL.cXM].axisRef.NcToPlc.ActPos>750))
	)
	AND GVL.bSafetyOn;

END_FUNCTION_BLOCK

// ---- POUs/StateMachine/StateTop/StateEnabled/FB_StateMaint.TcPOU
FUNCTION_BLOCK FB_StateMaint
VAR_IN_OUT
	stAxis  	: ARRAY [GVL.cXP .. GVL.cXM] OF ST_AxisGroup;
	bTopEntry	: BOOL;
END_VAR
VAR_INPUT
	eCommand			: E_Commands;
	stCalibrate			: ST_Calibrate;
	stChangeAxisEnable	: ST_ChangeAxisEnable;
	stChangeBrakeState	: ST_ChangeBrakeState;
	stClearAllFaults	: ST_ClearAllFaults;
	stClearAxisFaults	: ST_ClearAxisFaults;
	stDisableAllAxes	: ST_DisableAllAxes;
	stEnableAllAxes		: ST_EnableAllAxes;
	stGoToProd			: ST_GoToProd;
	stHomeAxis			: ST_HomeAxis;
	stMoveAxisAbsolute	: ST_MoveAxisAbsolute;
	stMoveAxisRelative	: ST_MoveAxisRelative;
END_VAR
VAR_OUTPUT
	bCalibDone		: BOOL;
	bMotionDone		: BOOL;
	stOutCalibDone	: ST_CalibDone;
	nSMState		: DINT;
END_VAR
VAR
	//state-machine
	eCurrentState	: E_StatesMaint;
	eNextState		: E_StatesMaint;
	fbHoming		: FB_Homing;
	fbCalibrating	: FB_StateCalibrating;
	fbMoving		: FB_StateMoving;
	fbStill			: FB_StateStill;
	bLowerEntry 	: BOOL;

	//other var
	eCopyCommand	: E_Commands;
	fbCalibRtrig	: R_TRIG;
	bCalibRestart : BOOL;
	
	//testVar
	//a, b, c : INT;
	
END_VAR


IF bTopEntry = TRUE THEN
	bTopEntry := FALSE;
	eNextState := E_StatesMaint.Still;
END_IF	
IF eCurrentState <> eNextState THEN
	bLowerEntry := TRUE;
END_IF
eCurrentState := eNextState;
nSMState := eCurrentState;
bMotionDone := FALSE;
//State Machine
CASE eCurrentState OF
	
	E_StatesMaint.Still:
		bCalibRestart := TRUE;
		fbStill(
			stAxis				:= stAxis, 
			bTopEntry			:= bLowerEntry, 
			eCommand			:= eCommand,
			stChangeAxisEnable 	:= stChangeAxisEnable,
			stChangeBrakeState	:= stChangeBrakeState,
			stClearAllFaults	:= stClearAllFaults,
			stClearAxisFaults	:= stClearAxisFaults,
			stDisableAllAxes	:= stDisableAllAxes,
			stEnableAllAxes		:= stEnableAllAxes);
		IF eCommand <> E_Commands.noCommand THEN (*checks if there is a new command*)
			IF eCommand = E_Commands.calibrate THEN
				eNextState := E_StatesMaint.Calibrating;
			ELSIF eCommand = E_Commands.closeShutter OR_ELSE
				eCommand = E_Commands.homeAxis OR_ELSE
				eCommand = E_Commands.moveAxisAbsolute OR_ELSE
				eCommand = E_Commands.moveAxisRelative THEN
					eCopyCommand := eCommand; (*need to copy since eCommand is only valid for 1 cycle. Resets to noCommand next cycle.*)
					eNextState := E_StatesMaint.Moving;
			END_IF
		END_IF
		//a := a+1;
	
	E_StatesMaint.Calibrating:
		bCalibDone := FALSE;
		fbHoming(stAxis:=stAxis, bTopEntry:=bLowerEntry);
		fbCalibRtrig(CLK:=(stAxis[GVL.cXP].axisRef.Status.Homed AND stAxis[GVL.cXM].axisRef.Status.Homed AND NOT fbHoming.bBusy));
		IF fbCalibRtrig.Q THEN
			bLowerEntry:=TRUE;
		END_IF
		fbCalibrating(stAxis:=stAxis, bTopEntry:=bLowerEntry, bCalibDone:=bCalibDone, bInterrupted:=bCalibRestart, stOutCalibDone=>stOutCalibDone);
		IF bCalibDone THEN
			eNextState := E_StatesMaint.Still;
		END_IF
		//b:=b+1;
		
	E_StatesMaint.Moving:
		fbMoving(
			stAxis				:= stAxis, 
			bTopEntry			:= bLowerEntry, 
			eCommand			:= eCopyCommand,
			stMoveAxisAbsolute 	:= stMoveAxisAbsolute,
			stMoveAxisRelative	:= stMoveAxisRelative);
		IF NOT fbMoving.bBusy THEN
			eNextState := E_StatesMaint.Still;
			bMotionDone := TRUE;
		END_IF
		//c:=c+1;
END_CASE

END_FUNCTION_BLOCK

// ---- POUs/StateMachine/StateTop/StateEnabled/StateMaint/FB_Homing.TcPOU
FUNCTION_BLOCK FB_Homing
VAR_IN_OUT
	stAxis  	: ARRAY [GVL.cXP .. GVL.cXM] OF ST_AxisGroup;
	bTopEntry	: BOOL;
END_VAR
VAR_OUTPUT
	bBusy : BOOL;
END_VAR
VAR
	//state-machine
	nCurrentState	: INT;
	nNextState		: INT;

	//other var
	fbHomeDelay		: TON;
	
	//testVar
	a,b,c :INT;
END_VAR

//////////////////////////////////////////////////
//Performs homing routine						//
//////////////////////////////////////////////////

IF bTopEntry = TRUE THEN
	bTopEntry := FALSE;
	nNextState := 410;
	bBusy := TRUE;
END_IF	
nCurrentState := nNextState;
CASE nCurrentState OF
	0:
	
	410: //Clear Homed flag and calibrated flag
		fbHomeDelay(IN:=FALSE);
		stAxis[GVL.cXP].mcHome(Axis := stAxis[GVL.cXP].axisRef, HomingMode := MC_ResetCalibration, bCalibrationCam := TRUE, Execute := TRUE);
		stAxis[GVL.cXM].mcHome(Axis := stAxis[GVL.cXM].axisRef, HomingMode := MC_ResetCalibration, bCalibrationCam := TRUE, Execute := TRUE);
		stAxis[GVL.cXP].bIsCalibrated := FALSE;
		stAxis[GVL.cXM].bIsCalibrated := FALSE;
		IF stAxis[GVL.cXP].mcHome.Done AND stAxis[GVL.cXM].mcHome.Done THEN
			stAxis[GVL.cXP].mcHome(Axis := stAxis[GVL.cXP].axisRef, Execute := FALSE);
			stAxis[GVL.cXM].mcHome(Axis := stAxis[GVL.cXM].axisRef, Execute := FALSE);
			nNextState := 420;
			a:=a+1;
		END_IF
		b:=b+1;
		
	420: //Scan for home switch
		stAxis[GVL.cXP].mcJog(Axis := stAxis[GVL.cXP].axisRef, Mode := MC_JOGMODE_CONTINOUS, Velocity := GVL.cScanVel, JogBackwards := NOT stAxis[GVL.cXP].bLimitHome);
		stAxis[GVL.cXM].mcJog(Axis := stAxis[GVL.cXM].axisRef, Mode := MC_JOGMODE_CONTINOUS, Velocity := GVL.cScanVel, JogForward := NOT stAxis[GVL.cXM].bLimitHome);
		IF stAxis[GVL.cXP].bLimitHome AND stAxis[GVL.cXM].bLimitHome THEN
			stAxis[GVL.cXP].mcJog(Axis := stAxis[GVL.cXP].axisRef, Mode := MC_JOGMODE_CONTINOUS, JogBackwards := FALSE);
			stAxis[GVL.cXM].mcJog(Axis := stAxis[GVL.cXM].axisRef, Mode := MC_JOGMODE_CONTINOUS, JogForward := FALSE);
			nNextState := 430;
		END_IF

	430: //back off from switch
		stAxis[GVL.cXP].mcJog(Axis := stAxis[GVL.cXP].axisRef, Mode := MC_JOGMODE_CONTINOUS, Velocity := GVL.cScanVel, JogForward := stAxis[GVL.cXP].bLimitHome);
		stAxis[GVL.cXM].mcJog(Axis := stAxis[GVL.cXM].axisRef, Mode := MC_JOGMODE_CONTINOUS, Velocity := GVL.cScanVel, JogBackwards := stAxis[GVL.cXM].bLimitHome);
		IF NOT stAxis[GVL.cXP].bLimitHome AND NOT stAxis[GVL.cXM].bLimitHome THEN
			stAxis[GVL.cXP].mcJog(Axis := stAxis[GVL.cXP].axisRef, Mode := MC_JOGMODE_CONTINOUS, JogForward := FALSE);
			stAxis[GVL.cXM].mcJog(Axis := stAxis[GVL.cXM].axisRef, Mode := MC_JOGMODE_CONTINOUS, JogBackwards := FALSE);
			nNextState := 440;
		END_IF
		
	440: //slowly homed back to switch
		stAxis[GVL.cXP].mcJog(Axis := stAxis[GVL.cXP].axisRef, Mode := MC_JOGMODE_CONTINOUS, Velocity := GVL.cHomeVel, JogBackwards := NOT stAxis[GVL.cXP].bLimitHome);
		stAxis[GVL.cXM].mcJog(Axis := stAxis[GVL.cXM].axisRef, Mode := MC_JOGMODE_CONTINOUS, Velocity := GVL.cHomeVel, JogForward := NOT stAxis[GVL.cXM].bLimitHome);
		IF stAxis[GVL.cXP].bLimitHome AND stAxis[GVL.cXM].bLimitHome THEN
			stAxis[GVL.cXP].mcJog(Axis := stAxis[GVL.cXP].axisRef, Mode := MC_JOGMODE_CONTINOUS, JogBackwards := FALSE);
			stAxis[GVL.cXM].mcJog(Axis := stAxis[GVL.cXM].axisRef, Mode := MC_JOGMODE_CONTINOUS, JogForward := FALSE);
			nNextState := 450;
		END_IF	

	450://delay
		fbHomeDelay(IN:=TRUE, PT:=T#100MS);
		IF fbHomeDelay.Q THEN
			fbHomeDelay(IN:=FALSE);	
			nNextState := 460;
		END_IF
		
	460://set home
		stAxis[GVL.cXP].mcHome(Axis := stAxis[GVL.cXP].axisRef, Position := GVL.cPosStart, HomingMode := MC_DIRECT, Execute := TRUE);
		stAxis[GVL.cXM].mcHome(Axis := stAxis[GVL.cXM].axisRef, Position := GVL.cPosEnd, HomingMode := MC_DIRECT, Execute := TRUE);	
		IF stAxis[GVL.cXP].mcHome.Done AND stAxis[GVL.cXM].mcHome.Done THEN
			stAxis[GVL.cXP].mcHome(Axis := stAxis[GVL.cXP].axisRef, Execute := FALSE);
			stAxis[GVL.cXM].mcHome(Axis := stAxis[GVL.cXM].axisRef, Execute := FALSE);
			nNextState := 470;
		END_IF	
		
	470://delay
		fbHomeDelay(IN:=TRUE, PT:=T#100MS);
		IF fbHomeDelay.Q THEN
			fbHomeDelay(IN:=FALSE);	
			nNextState := 480;
		END_IF
		
	480: //End Action
		bBusy := FALSE;
		nNextState :=0;
END_CASE

END_FUNCTION_BLOCK

// ---- POUs/StateMachine/StateTop/StateEnabled/StateMaint/FB_StateCalibrating.TcPOU
FUNCTION_BLOCK FB_StateCalibrating
VAR_IN_OUT
	stAxis  	: ARRAY [GVL.cXP .. GVL.cXM] OF ST_AxisGroup;	
	bTopEntry	: BOOL;
	bCalibDone	: BOOL;
	bInterrupted: BOOL;
END_VAR
VAR_OUTPUT
	stOutCalibDone	: ST_CalibDone;
END_VAR
VAR
	nCurrentState	: INT;
	nNextState		: INT;
	
	//counter
	i	: INT;
	nTripCountXP	: INT;
	nTripCountXM	: INT;
	
	//test var
	//a, b, c : INT;
END_VAR

//////////////////////////////////////////////////
//perform software calibration of axis. 		//
//////////////////////////////////////////////////
IF bInterrupted THEN
	bInterrupted := FALSE;
	nNextState := 0;
END_IF
IF bTopEntry = TRUE THEN
	bTopEntry := FALSE;
	nNextState :=8010;
END_IF	
nCurrentState := nNextState;
bCalibDone := FALSE;
CASE nCurrentState OF
	0:
	
	(*Perform software calibration of axis xp*)
	8010: //Clear previous Calibration value
		FOR i:=0 TO GVL.cTripCount BY 1 DO
			stAxis[GVL.cXP].fHallPosCal[0,i]:=0;
			stAxis[GVL.cXP].fHallPosCal[1,i]:=0;
		END_FOR
		stAxis[GVL.cXP].mcMoveAbs(Axis:=stAxis[GVL.cXP].axisRef, Execute:=FALSE);
		stAxis[GVL.cXM].mcMoveAbs(Axis:=stAxis[GVL.cXM].axisRef, Execute:=FALSE);
		stAxis[GVL.cXP].nTripCount := 0;	
		nTripCountXP := 0;	
		stAxis[GVL.cXP].bIsCalibrated := FALSE;
		nNextState:=8020;
		
	8020: //Put Shutter in Open Position
		stAxis[GVL.cXP].mcMoveAbs(Axis:=stAxis[GVL.cXP].axisRef, Position:=GVL.cPosStart, Velocity:=GVL.cPositionVel, Acceleration:=0, Deceleration:=0, Jerk:=0, Execute:=TRUE);
		stAxis[GVL.cXM].mcMoveAbs(Axis:=stAxis[GVL.cXM].axisRef, Position:=GVL.cPosEnd, Velocity:=GVL.cPositionVel, Acceleration:=0, Deceleration:=0, Jerk:=0, Execute:=TRUE);
		IF stAxis[GVL.cXP].mcMoveAbs.Done AND stAxis[GVL.cXM].mcMoveAbs.Done THEN
			stAxis[GVL.cXP].mcMoveAbs(Axis:=stAxis[GVL.cXP].axisRef, Execute:=FALSE);
			stAxis[GVL.cXM].mcMoveAbs(Axis:=stAxis[GVL.cXM].axisRef, Execute:=FALSE);
			nNextState:=8030;
		END_IF
		

	8030: //Calibrate AxisXP towards X- side.
		//record position and sequence of hall trips at rising and falling edge.
		FOR i:=GVL.cHallLower TO GVL.cHallUpper BY 1 DO
			IF GVL.nNumOfInputs[i].0 THEN
				//identifies which hall switch tripped along with if it's rising or falling edge
				stAxis[GVL.cXP].stHall[GVL.cDirPos, nTripCountXP].nSeq := INT_TO_WORD((i*10)+5);
				stAxis[GVL.cXP].stHall[GVL.cDirPos, nTripCountXP].bEdge := GVL.bInputEventState[i];
				stAxis[GVL.cXP].fHallPosCal[GVL.cDirPos, nTripCountXP] := stAxis[GVL.cXP].axisRef.NcToPlc.ActPos;
				nTripCountXP := nTripCountXP + 1;
			END_IF
		END_FOR
		//start moving axisXP towards x- side
		stAxis[GVL.cXP].mcMoveAbs(Axis:=stAxis[GVL.cXP].axisRef, Position:=GVL.cPosEnd, Velocity:=GVL.cCalibrateVel, Acceleration:=0, Deceleration:=0, Jerk:=0, Execute:=TRUE);
		IF stAxis[GVL.cXP].mcMoveAbs.Done THEN
			stAxis[GVL.cXP].mcMoveAbs(Axis:=stAxis[GVL.cXP].axisRef, Execute:=FALSE);
			nNextState:= 8040;
		END_IF
	
	8040: //Calibrate AxisXP towards X+ side.
		//record position and sequence of hall trips at rising and falling edge
		FOR i:=GVL.cHallLower TO GVL.cHallUpper BY 1 DO
			IF GVL.nNumOfInputs[i].0 THEN
				//identifies which hall switch tripped along with if it's rising or falling edge
				stAxis[GVL.cXP].stHall[GVL.cDirNeg, nTripCountXP].nSeq := INT_TO_WORD((i*10)+5);
				stAxis[GVL.cXP].stHall[GVL.cDirNeg, nTripCountXP].bEdge := GVL.bInputEventState[i];
				
				stAxis[GVL.cXP].fHallPosCal[GVL.cDirNeg, nTripCountXP] := stAxis[GVL.cXP].axisRef.NcToPlc.ActPos;
				nTripCountXP := nTripCountXP - 1;	
			
			END_IF
		END_FOR
		//start moving axisXP towards x+ side
		stAxis[GVL.cXP].mcMoveAbs(Axis:=stAxis[GVL.cXP].axisRef, Position:=GVL.cPosStart-0.1, Velocity:=GVL.cCalibrateVel, Acceleration:=0, Deceleration:=0, Jerk:=0, Execute:=TRUE);
		IF stAxis[GVL.cXP].mcMoveAbs.Done THEN
			stAxis[GVL.cXP].mcMoveAbs(Axis:=stAxis[GVL.cXP].axisRef, Execute:=FALSE);
			nNextState := 8050;
		END_IF
	
	8050: //move blade off switch to start tracking
		stAxis[GVL.cXP].mcJog(Axis := stAxis[GVL.cXP].axisRef, Mode := MC_JOGMODE_CONTINOUS, Velocity := GVL.cScanVel, JogForward := stAxis[GVL.cXP].bLimitHome);
		IF NOT stAxis[GVL.cXP].bLimitHome THEN
			stAxis[GVL.cXP].mcJog(Axis := stAxis[GVL.cXM].axisRef, Mode := MC_JOGMODE_CONTINOUS, JogForward := FALSE);
			nNextState := 8060;
		END_IF
		
	8060: //slowly home back to limit switch
		stAxis[GVL.cXP].mcJog(Axis := stAxis[GVL.cXP].axisRef, Mode := MC_JOGMODE_CONTINOUS, Velocity := GVL.cHomeVel, JogBackwards := NOT stAxis[GVL.cXP].bLimitHome);
		//a := a +1;
		IF stAxis[GVL.cXP].bLimitHome THEN
			//b := b+1;
			stAxis[GVL.cXP].mcJog(Axis := stAxis[GVL.cXP].axisRef, Mode := MC_JOGMODE_CONTINOUS, JogBackwards := FALSE);
			IF nTripCountXP = 0 THEN	
				stAxis[GVL.cXP].bIsCalibrated := TRUE; //should signal a warning to indicate bad calibration... Can be added later.
			END_IF
			nNextState := 9010;
		END_IF			
		

	(*Perform software calibration of axis xm*)
	9010: //Clear previous Calibration value
		FOR i:=0 TO GVL.cTripCount BY 1 DO
			stAxis[GVL.cXM].fHallPosCal[0,i]:=0;
			stAxis[GVL.cXM].fHallPosCal[1,i]:=0;
		END_FOR
		stAxis[GVL.cXM].nTripCount := 0;	
		nTripCountXM := 0;
		stAxis[GVL.cXM].bIsCalibrated := FALSE;
		nNextState:=9020;
		
	9020: //Put Shutter in Open Position
		stAxis[GVL.cXP].mcMoveAbs(Axis:=stAxis[GVL.cXP].axisRef, Position:=GVL.cPosStart, Velocity:=GVL.cPositionVel, Acceleration:=0, Deceleration:=0, Jerk:=0, Execute:=TRUE);
		stAxis[GVL.cXM].mcMoveAbs(Axis:=stAxis[GVL.cXM].axisRef, Position:=GVL.cPosEnd, Velocity:=GVL.cPositionVel, Acceleration:=0, Deceleration:=0, Jerk:=0, Execute:=TRUE);
		IF stAxis[GVL.cXP].mcMoveAbs.Done AND stAxis[GVL.cXM].mcMoveAbs.Done THEN
			stAxis[GVL.cXP].mcMoveAbs(Axis:=stAxis[GVL.cXP].axisRef, Execute:=FALSE);
			stAxis[GVL.cXM].mcMoveAbs(Axis:=stAxis[GVL.cXM].axisRef, Execute:=FALSE);
			nNextState:=9030;
		END_IF
	
	9030: //Calibrate stAxisGVL.cXM twoards X+ side.
		//record position and sequence of hall trips at rising and falling edge.
		FOR i:=GVL.cHallLower TO GVL.cHallUpper BY 1 DO
			IF GVL.nNumOfInputs[i].0 THEN
				//identifies which hall switch tripped along with if it's rising or falling edge
				stAxis[GVL.cXM].stHall[GVL.cDirNeg, nTripCountXM].nSeq := INT_TO_WORD((i*10)+5);
				stAxis[GVL.cXM].stHall[GVL.cDirNeg, nTripCountXM].bEdge := GVL.bInputEventState[i];
				
				stAxis[GVL.cXM].fHallPosCal[GVL.cDirNeg, nTripCountXM] := stAxis[GVL.cXM].axisRef.NcToPlc.ActPos;
				nTripCountXM := nTripCountXM + 1;	
			END_IF
		END_FOR
		//start moving stAxisGVL.cXP towards x+ side
		stAxis[GVL.cXM].mcMoveAbs(Axis:=stAxis[GVL.cXM].axisRef, Position:=GVL.cPosStart, Velocity:=GVL.cCalibrateVel, Acceleration:=0, Deceleration:=0, Jerk:=0, Execute:=TRUE);
		IF stAxis[GVL.cXM].mcMoveAbs.Done THEN
			stAxis[GVL.cXM].mcMoveAbs(Axis:=stAxis[GVL.cXP].axisRef, Execute:=FALSE);
			nNextState:= 9040;
		END_IF
	
	
	9040: //Calibrate stAxisGVL.cXM twoards X- side.
		//record position and sequence of hall trips at rising and falling edge.
		FOR i:=GVL.cHallLower TO GVL.cHallUpper BY 1 DO
			IF GVL.nNumOfInputs[i].0 THEN
				//identifies which hall switch tripped along with if it's rising or falling edge
				stAxis[GVL.cXM].stHall[GVL.cDirPos, nTripCountXM].nSeq := INT_TO_WORD((i*10)+5);
				stAxis[GVL.cXM].stHall[GVL.cDirPos, nTripCountXM].bEdge := GVL.bInputEventState[i];
				
				stAxis[GVL.cXM].fHallPosCal[GVL.cDirPos, nTripCountXM] := stAxis[GVL.cXM].axisRef.NcToPlc.ActPos;
				nTripCountXM := nTripCountXM - 1;	
			END_IF
		END_FOR
		//start moving stAxisGVL.cXP towards x- side
		stAxis[GVL.cXM].mcMoveAbs(Axis:=stAxis[GVL.cXM].axisRef, Position:=GVL.cPosEnd+0.1, Velocity:=GVL.cCalibrateVel, Acceleration:=0, Deceleration:=0, Jerk:=0, Execute:=TRUE);
		IF stAxis[GVL.cXM].mcMoveAbs.Done THEN
			stAxis[GVL.cXM].mcMoveAbs(Axis:=stAxis[GVL.cXM].axisRef, Execute:=FALSE);
			nNextState := 9050;
		END_IF
		
	9050: //move blade off switch to start tracking 
		stAxis[GVL.cXM].mcJog(Axis:=stAxis[GVL.cXM].axisRef, Mode:=MC_JOGMODE_CONTINOUS, Velocity:=GVL.cScanVel, JogBackwards:=stAxis[GVL.cXM].bLimitHome);
		IF NOT stAxis[GVL.cXM].bLimitHome THEN
			stAxis[GVL.cXM].mcJog(Axis:=stAxis[GVL.cXM].axisRef, Mode:=MC_JOGMODE_CONTINOUS, JogBackwards:=FALSE);
			nNextState := 9060;
		END_IF

	9060: //slowly homed back to switch
		stAxis[GVL.cXM].mcJog(Axis:=stAxis[GVL.cXM].axisRef, Mode:=MC_JOGMODE_CONTINOUS, Velocity:=GVL.cHomeVel, JogForward := NOT stAxis[GVL.cXM].bLimitHome);
		IF stAxis[GVL.cXM].bLimitHome THEN
			stAxis[GVL.cXM].mcJog(Axis := stAxis[GVL.cXM].axisRef, Mode := MC_JOGMODE_CONTINOUS, JogForward := FALSE);
				IF nTripCountXM=0 THEN
					stAxis[GVL.cXM].bIsCalibrated := TRUE;  //should signal a warning to indicate bad calibration... Can be added later.
				END_IF
			nNextState := 9070;
		END_IF			
		
	9070: //save calibration data to stOutCalibDone to be sent to CCS
		FOR i:=0 TO GVL.cTripCount BY 1 DO
			stOutCalibDone.hallPosCal[GVL.cXP, GVL.cDirPos, i] := stAxis[GVL.cXP].fHallPosCal[GVL.cDirPos, i];
			stOutCalibDone.hallPosCal[GVL.cXP, GVL.cDirNeg, i] := stAxis[GVL.cXP].fHallPosCal[GVL.cDirNeg, i];
			stOutCalibDone.hallPosCal[GVL.cXM, GVL.cDirPos, i] := stAxis[GVL.cXM].fHallPosCal[GVL.cDirPos, i];
			stOutCalibDone.hallPosCal[GVL.cXM, GVL.cDirNeg, i] := stAxis[GVL.cXM].fHallPosCal[GVL.cDirNeg, i];
		END_FOR
		bCalibDone := TRUE;
		nNextState :=0;
	
END_CASE

END_FUNCTION_BLOCK

// ---- POUs/StateMachine/StateTop/StateEnabled/StateMaint/FB_StateMoving.TcPOU
FUNCTION_BLOCK FB_StateMoving
VAR_IN_OUT
	stAxis  	: ARRAY [GVL.cXP .. GVL.cXM] OF ST_AxisGroup;
	bTopEntry	: BOOL;
	eCommand	: E_Commands;
END_VAR
VAR_INPUT
	stHomeAxis			: ST_HomeAxis;
	stMoveAxisAbsolute	: ST_MoveAxisAbsolute;
	stMoveAxisRelative	: ST_MoveAxisRelative;
END_VAR
VAR_OUTPUT
	bBusy		: BOOL;
END_VAR
VAR
	//state-machine
	nCurrentState	: INT;
	nNextState		: INT;
	bLowerEntry 	: BOOL;
	//homing subroutine
	fbHoming	: FB_Homing;
	//move relative vars
	fDistance, fTime, fSpeed, fAccel, fJerk : LREAL;

END_VAR

IF bTopEntry = TRUE THEN
	bTopEntry := FALSE;
	IF eCommand = E_Commands.homeAxis THEN
		nNextState := 1000;
	ELSIF eCommand = E_Commands.moveAxisAbsolute THEN
		fDistance := ABS(stAxis[stMoveAxisAbsolute.axisIndex].axisRef.NcToPlc.ActPos - stMoveAxisAbsolute.position);
		fSpeed	:= stMoveAxisAbsolute.speed;
		IF (fSpeed>0) THEN
			IF (fSpeed>1668.355556) THEN
				fSpeed:=1668.355556;
			END_IF
			fTime 	:= (2*fDistance)/(fSpeed);
			IF (fTime<0.9) THEN
				fTime:=0.9;
			END_IF
			fAccel 	:= (8*fDistance)/(fTime*fTime);
			fJerk	:= (32*fDistance)/(fTime*fTime*fTime);
		END_IF
		nNextState := 1010;
	ELSIF eCommand = E_Commands.moveAxisRelative THEN
		(* 
			equations  		(distance in mm, time in sec)
			Velocity 		= 2*distance/time
			Acceleration 	= 8*distance/time^2
			jerk 			= 32*distance/time^3
		*)
		fTime	:= TIME_TO_LREAL(stMoveAxisRelative.moveTime)/1000;
		IF (fTime>0) THEN
			fSpeed 	:= (2*ABS(stMoveAxisRelative.distance))/(fTime);
			fAccel 	:= (8*ABS(stMoveAxisRelative.distance))/(fTime*fTime);
			fJerk	:= (32*ABS(stMoveAxisRelative.distance))/(fTime*fTime*fTime);
		END_IF

		nNextState := 1020;
	END_IF
END_IF	

IF (fSpeed > 1668.35556) THEN
	fSpeed := 1668.3556;
END_IF
IF (fAccel > 7414.91358) THEN
	fAccel := 7414.91358;
END_IF
IF (fJerk > 32955.17147) THEN
	fJerk := 32955.17147;
END_IF

IF nCurrentState <> nNextState THEN
	bLowerEntry := TRUE;
END_IF
nCurrentState := nNextState;
bBusy := TRUE;
CASE nCurrentState OF
		
	1000://Homing routine
		fbHoming(stAxis:=stAxis, bTopEntry:=bLowerEntry);
		IF NOT fbHoming.bBusy THEN
			nNextState := 2000;
		END_IF
		
	1010://move absolute
		stAxis[stMoveAxisAbsolute.axisIndex].mcMoveAbs(Axis:=stAxis[stMoveAxisAbsolute.axisIndex].axisRef,
			Position:=stMoveAxisAbsolute.position, Velocity:=fSpeed, Acceleration:= fAccel, Deceleration:= fAccel, Jerk:= fJerk,  Execute:=TRUE);
		IF stAxis[stMoveAxisAbsolute.axisIndex].mcMoveAbs.Done THEN
			stAxis[stMoveAxisAbsolute.axisIndex].mcMoveAbs(Axis:=stAxis[stMoveAxisAbsolute.axisIndex].axisRef, Execute:=FALSE);
			nNextState := 2000;
		END_IF
		
	1020://move relative with different motion profile parameter
		stAxis[stMoveAxisRelative.axisIndex].mcMoveRel(Axis:=stAxis[stMoveAxisRelative.axisIndex].axisRef,
			Distance:=stMoveAxisRelative.distance, Velocity:=fSpeed, Acceleration:=fAccel, Jerk:=fJerk, Execute:=TRUE);
		IF stAxis[stMoveAxisRelative.axisIndex].mcMoveRel.Done THEN
			stAxis[stMoveAxisRelative.axisIndex].mcMoveRel(Axis:=stAxis[stMoveAxisRelative.axisIndex].axisRef, Execute:=FALSE);
			nNextState := 2000;
		END_IF
			
	2000:
		bBusy := FALSE;
	
END_CASE

END_FUNCTION_BLOCK

// ---- POUs/StateMachine/StateTop/StateEnabled/StateMaint/FB_StateStill.TcPOU
FUNCTION_BLOCK FB_StateStill
VAR_IN_OUT
	stAxis  	: ARRAY [GVL.cXP .. GVL.cXM] OF ST_AxisGroup;
	bTopEntry	: BOOL;
END_VAR
VAR_INPUT
	eCommand			: E_Commands;
	stChangeAxisEnable	: ST_ChangeAxisEnable;
	stChangeBrakeState	: ST_ChangeBrakeState;
	stClearAllFaults	: ST_ClearAllFaults;
	stClearAxisFaults	: ST_ClearAxisFaults;
	stDisableAllAxes	: ST_DisableAllAxes;
	stEnableAllAxes		: ST_EnableAllAxes;
END_VAR
VAR_OUTPUT
	bBusy	: BOOL;
END_VAR
VAR
	//state-machine
	nCurrentState	: INT;
	nNextState		: INT;
END_VAR


IF bTopEntry = TRUE THEN
	bTopEntry := FALSE;
	bBusy := TRUE;
END_IF	

IF eCommand = E_Commands.clearAllFaults THEN
	nNextState := 1000;
ELSIF eCommand = E_Commands.changeAxisEnable THEN
	nNextState := 1010	;
ELSIF eCommand = E_Commands.clearAxisFaults THEN
	nNextState := 1020;
ELSIF eCommand = E_Commands.enableAllAxes THEN
	nNextState := 1030;
ELSIF eCommand = E_Commands.disableAllAxes THEN
	nNextState := 1040;
ELSIF eCommand = E_Commands.changeBrakeState THEN
	nNextState := 1050;
END_IF

nCurrentState := nNextState;

CASE nCurrentState OF

	1000:
		stAxis[GVL.cXM].mcReset(Axis:=stAxis[GVL.cXM].axisRef, Execute:=TRUE);
		stAxis[GVL.cXM].mcReset(Axis:=stAxis[GVL.cXM].axisRef, Execute:=TRUE);
		IF stAxis[GVL.cXP].mcReset.Done AND stAxis[GVL.cXM].mcReset.Done THEN
			stAxis[GVL.cXM].mcReset(Axis:=stAxis[GVL.cXM].axisRef, Execute:=FALSE);
			stAxis[GVL.cXM].mcReset(Axis:=stAxis[GVL.cXM].axisRef, Execute:=FALSE);
			nNextState := 2000; 
		END_IF
		
	1010:	
		stAxis[stChangeAxisEnable.axisIndex].mcPower(Axis:=stAxis[stChangeAxisEnable.axisIndex].axisRef,
			 Enable:=stChangeAxisEnable.enabled, Enable_Positive:=stChangeAxisEnable.enabled, Enable_Negative:=stChangeAxisEnable.enabled);
		//nNextState := 2000; 

	1020:	
		stAxis[stClearAxisFaults.axisIndex].mcReset(Axis:=stAxis[stClearAxisFaults.axisIndex].axisRef, Execute:=TRUE);
		IF stAxis[stClearAxisFaults.axisIndex].mcReset.Done THEN
			stAxis[stClearAxisFaults.axisIndex].mcReset(Axis:=stAxis[stClearAxisFaults.axisIndex].axisRef, Execute:=FALSE);
			nNextState := 2000; 
		END_IF

	1030:
		stAxis[GVL.cXP].mcPower(Axis:=stAxis[GVL.cXP].axisRef, Enable:=TRUE, Enable_Positive:=TRUE, Enable_Negative:=TRUE);
		stAxis[GVL.cXM].mcPower(Axis:=stAxis[GVL.cXM].axisRef, Enable:=TRUE, Enable_Positive:=TRUE, Enable_Negative:=TRUE);
		nNextState := 2000; 

	1040:	
		stAxis[GVL.cXP].mcPower(Axis:=stAxis[GVL.cXP].axisRef, Enable:=FALSE, Enable_Positive:=FALSE, Enable_Negative:=FALSE);
		stAxis[GVL.cXM].mcPower(Axis:=stAxis[GVL.cXM].axisRef, Enable:=FALSE, Enable_Positive:=FALSE, Enable_Negative:=FALSE);
		nNextState := 2000; 
		
	1050:
		stAxis[stChangeBrakeState.axisIndex].bBrake := NOT stChangeBrakeState.state;
		nNextState := 2000; 

	2000:
		bBusy := FALSE;
	
END_CASE

END_FUNCTION_BLOCK

// ---- POUs/StateMachine/StateTop/StateEnabled/FB_StateProd.TcPOU
FUNCTION_BLOCK FB_StateProd
VAR_IN_OUT
	stAxis  	: ARRAY [GVL.cXP .. GVL.cXM] OF ST_AxisGroup;	
	bTopEntry	: BOOL;
END_VAR
VAR_INPUT
	eCommand		: E_Commands;
	fSpeed			: LREAL;
	stOpenShutter	: ST_OpenShutter;
	stCloseShutter	: ST_CloseShutter;
	stTakeExposure	: ST_TakeExposure;
END_VAR
VAR_OUTPUT
	bMotionDone		: BOOL;
	stOutTimer		: ST_Timer;
	
	nSMState		: DINT;
END_VAR
VAR
	//motion parameter
	fTime			: LREAL;
	fAccel			: LREAL;
	fJerk			: LREAL;
	
	//state-machine
	eCurrentState	: E_StatesProd;
	eNextState		: E_StatesProd;
	fbClosed		: FB_StateClosed;
	fbClosing		: FB_StateClosing;
	fbOpened		: FB_StateOpened;
	fbOpening		: FB_StateOpening;
	fbTravelling	: FB_StateTravelling;
	bLowerEntry	: BOOL;

	//shutter blade
	nRet	: INT;
	nExt	: INT;
	
	//Taking Exposure Variable
	bTakingExposure	: BOOL;
	fbExpoTimer		:  TON;
	
END_VAR


IF bTopEntry = TRUE THEN
	bTopEntry := FALSE;
	eNextState := E_StatesProd.Closed;
	(*These values are opposite of what they should be but they are going to be swapped to correct value as the state machine enter "Closed" state*)
	IF (stAxis[GVL.cXP].axisRef.NcToPlc.ActPos<1) AND (stAxis[GVL.cXM].axisRef.NcToPlc.ActPos<1) THEN
		nRet := GVL.cXP;
		nExt := GVL.cXM;
	END_IF
	IF (stAxis[GVL.cXP].axisRef.NcToPlc.ActPos>750) AND (stAxis[GVL.cXM].axisRef.NcToPlc.ActPos>750) THEN
		nRet := GVL.cXM;
		nExt := GVL.cXP;
	END_IF
	bLowerEntry := TRUE;
END_IF	

(* calculate acceleration and jerk *)
IF (fSpeed>0) THEN
	IF (fSpeed>1668.355556) THEN
		fSpeed:=1668.355556;
	END_IF
	fTime	:= 2*GVL.cPosEnd/fSpeed;
	IF (fTime<0.9) THEN
		fTime:=0.9;
	END_IF
	fAccel 	:= (8*GVL.cPosEnd)/(fTime*fTime);
	fJerk	:= (32*GVL.cPosEnd)/(fTime*fTime*fTime);
END_IF

IF eCurrentState <> eNextState THEN
	bLowerEntry := TRUE;
END_IF

eCurrentState := eNextState;
nSMState := eCurrentState;
fbExpoTimer(IN:=bTakingExposure, PT:=stTakeExposure.exposureTime);
bMotionDone := FALSE;

CASE eCurrentState OF
	
	E_StatesProd.Closed:
		fbClosed(stAxis:=stAxis, bTopEntry:=bLowerEntry, nRet:=nRet, nExt:=nExt);
		bTakingExposure := FALSE;
		IF eCommand = E_Commands.openShutter OR eCommand = E_Commands.takeExposure THEN
			IF eCommand = E_Commands.takeExposure THEN
				bTakingExposure := TRUE;
			END_IF
			eNextState := E_StatesProd.Opening;
		END_IF

	E_StatesProd.Opening:
		fbOpening(stAxis:=stAxis, bTopEntry:=bLowerEntry, fSpeed:=fSpeed, fAccel:=fAccel, fJerk:=fJerk, nRet:=nRet);
		IF NOT fbOpening.bBusy THEN
			bMotionDone := TRUE;
			eNextState := E_StatesProd.Opened;
		END_IF
		IF fbExpoTimer.Q THEN 
			eNextState := E_StatesProd.Traveling;
			stOutTimer.sequence:=stOutTimer.sequence+1;
		END_IF
	
	E_StatesProd.Opened:
		fbOpened(stAxis:=stAxis, bTopEntry:=bLowerEntry);
		IF eCommand = E_Commands.closeShutter OR fbExpoTimer.Q THEN
			IF fbExpoTimer.Q THEN
				stOutTimer.sequence:=stOutTimer.sequence+1;
			END_IF
			eNextState := E_StatesProd.Closing;
			(*add error code or warning if timer is active and closeShutter command is issued*)
		END_IF
		
	E_StatesProd.Closing:
		fbClosing(stAxis:=stAxis, bTopEntry:=bLowerEntry, nExt:=nExt, fSpeed:=fSpeed, fAccel:=fAccel, fJerk:=fJerk);
		IF NOT fbClosing.bBusy THEN
			bMotionDone := TRUE;
			eNextState := E_StatesProd.Closed;
		END_IF
	
	E_StatesProd.Traveling:
		fbTravelling(stAxis:=stAxis, bTopEntry:=bLowerEntry, nExt:=nExt, nRet:=nRet, fSpeed:=fspeed, fAccel:=fAccel, fJerk:=fJerk);
		IF NOT fbTravelling.bBusy THEN
			bMotionDone := TRUE;
			eNextState := E_StatesProd.Closing;
		END_IF
	
END_CASE

END_FUNCTION_BLOCK

// ---- POUs/StateMachine/StateTop/StateEnabled/StateProd/FB_StateClosed.TcPOU
FUNCTION_BLOCK FB_StateClosed
VAR_IN_OUT
	stAxis  	: ARRAY [GVL.cXP .. GVL.cXM] OF ST_AxisGroup;	
	bTopEntry	: BOOL;
	nRet	: INT;
	nExt	: INT;
END_VAR

VAR
	nCurrentState	: INT;
	nNextState		: INT;
END_VAR



IF bTopEntry = TRUE THEN
	bTopEntry := FALSE;
	nRet := 1 - nRet;
	nExt := 1 - nExt;
	nNextState := 1000;
END_IF	
nCurrentState := nNextState;

CASE nCurrentState OF

	1000:


END_CASE

END_FUNCTION_BLOCK

// ---- POUs/StateMachine/StateTop/StateEnabled/StateProd/FB_StateClosing.TcPOU
FUNCTION_BLOCK FB_StateClosing
VAR_IN_OUT
	stAxis 	 	: ARRAY [GVL.cXP .. GVL.cXM] OF ST_AxisGroup;	
	bTopEntry	: BOOL;
END_VAR
VAR_INPUT
	nExt	: INT;
	fSpeed	: LREAL;
	fAccel	: LREAL;
	fJerk	: LREAL;
END_VAR
VAR_OUTPUT
	bBusy	: BOOL;
END_VAR
VAR
	//state-machine
	nCurrentState	: INT;
	nNextState		: INT;
END_VAR

//////////////////////////////////////////////////
//Closes shutter								//
//////////////////////////////////////////////////
IF bTopEntry = TRUE THEN
	bTopEntry := FALSE;
	nNextState := 1300;
END_IF

bBusy := TRUE;
nCurrentState := nNextState;

CASE nCurrentState OF
	
(*Perform Open Shutter Motion*)
	1300:
		IF nExt = GVL.cXP THEN
			stAxis[GVL.cXP].mcMoveAbs(Axis:=stAxis[GVL.cXP].axisRef, Position:=GVL.cPosEnd, Velocity:=fSpeed, Acceleration:=fAccel, Deceleration:=fAccel, Jerk:=fJerk, Execute:=TRUE);
		ELSIF nExt = GVL.cXM THEN	
			stAxis[GVL.cXM].mcMoveAbs(Axis:=stAxis[GVL.cXM].axisRef, Position:=GVL.cPosStart, Velocity:=fSpeed, Acceleration:=fAccel, Deceleration:=fAccel, Jerk:=fJerk, Execute:=TRUE);
		END_IF
		IF stAxis[GVL.cXP].mcMoveAbs.Done OR stAxis[GVL.cXM].mcMoveAbs.Done THEN
			stAxis[GVL.cXP].mcMoveAbs(Axis:=stAxis[GVL.cXP].axisRef, Execute:=FALSE);
			stAxis[GVL.cXM].mcMoveAbs(Axis:=stAxis[GVL.cXM].axisRef, Execute:=FALSE);
			nNextState := 1310;
		END_IF	
		
	1310: //End action
		bBusy := FALSE;

END_CASE

END_FUNCTION_BLOCK

// ---- POUs/StateMachine/StateTop/StateEnabled/StateProd/FB_StateOpened.TcPOU
FUNCTION_BLOCK FB_StateOpened
VAR_IN_OUT
	stAxis  	: ARRAY [GVL.cXP .. GVL.cXM] OF ST_AxisGroup;	
	bTopEntry	: BOOL;
END_VAR
VAR
	//state-machine
	nCurrentState	: INT;
	nNextState		: INT;
END_VAR


IF bTopEntry = TRUE THEN
	bTopEntry := FALSE;
	nNextState := 1200;
END_IF	
nCurrentState := nNextState;

CASE nCurrentState OF
	1200:

END_CASE

END_FUNCTION_BLOCK

// ---- POUs/StateMachine/StateTop/StateEnabled/StateProd/FB_StateOpening.TcPOU
FUNCTION_BLOCK FB_StateOpening
VAR_IN_OUT
	stAxis  	: ARRAY [GVL.cXP .. GVL.cXM] OF ST_AxisGroup;	
	bTopEntry	: BOOL;
END_VAR
VAR_INPUT
	nRet	: INT;
	fSpeed	: LREAL;
	fAccel	: LREAL;
	fJerk	: LREAL;
END_VAR
VAR_OUTPUT
	bBusy	: BOOL;
END_VAR
VAR
	//state-machine
	nCurrentState	: INT;
	nNextState		: INT;
	
END_VAR

//////////////////////////////////////////////////
//Puts shutter in open position					//
//////////////////////////////////////////////////
IF bTopEntry = TRUE THEN
	bTopEntry 	:= FALSE;
	nNextState 	:= 1100;
END_IF
bBusy 	:= TRUE;
nCurrentState 	:= nNextState;

CASE nCurrentState OF
(*Perform Open Shutter Motion*)
	1100:
		IF nRet = GVL.cXP THEN
			stAxis[GVL.cXP].mcMoveAbs(Axis:=stAxis[GVL.cXP].axisRef, Position:=GVL.cPosStart, Velocity:=fSpeed, Acceleration:=fAccel, Deceleration:=fAccel, Jerk:=fJerk, Execute:=TRUE);
		ELSIF nRet = GVL.cXM THEN	
			stAxis[GVL.cXM].mcMoveAbs(Axis:=stAxis[GVL.cXM].axisRef, Position:=GVL.cPosEnd, Velocity:=fSpeed, Acceleration:=fAccel, Deceleration:=fAccel, Jerk:=fJerk, Execute:=TRUE);
		END_IF
		IF stAxis[GVL.cXP].mcMoveAbs.Done OR stAxis[GVL.cXM].mcMoveAbs.Done THEN
			stAxis[GVL.cXP].mcMoveAbs(Axis:=stAxis[GVL.cXP].axisRef, Execute:=FALSE);
			stAxis[GVL.cXM].mcMoveAbs(Axis:=stAxis[GVL.cXM].axisRef, Execute:=FALSE);
			nNextState := 1110;
		END_IF	
		
	1110: //End action
		bBusy := FALSE;

END_CASE

END_FUNCTION_BLOCK

// ---- POUs/StateMachine/StateTop/StateEnabled/StateProd/FB_StateTravelling.TcPOU
FUNCTION_BLOCK FB_StateTravelling
VAR_IN_OUT
	stAxis 	 	: ARRAY [GVL.cXP .. GVL.cXM] OF ST_AxisGroup;	
	bTopEntry	: BOOL;
END_VAR
VAR_INPUT
	nExt	: INT;
	nRet	: INT;
	fSpeed	: LREAL;
	fAccel	: LREAL;
	fJerk	: LREAL;
END_VAR
VAR_OUTPUT
	bBusy	: BOOL;
END_VAR
VAR
	//state-machine
	nCurrentState	: INT;
	nNextState		: INT;
END_VAR



IF bTopEntry = TRUE THEN
	bTopEntry := FALSE;
	nNextState := 1400;
END_IF

bBusy := TRUE;
nCurrentState := nNextState;

CASE nCurrentState OF
	
(*Perform Open Shutter Motion*)
	1400:
		IF nRet = GVL.cXP THEN
			stAxis[GVL.cXP].mcMoveAbs(Axis:=stAxis[GVL.cXP].axisRef, Position:=GVL.cPosStart, Velocity:=fSpeed, Acceleration:=fAccel, Deceleration:=fAccel, Jerk:=fJerk, Execute:=TRUE);
		ELSIF nRet = GVL.cXM THEN
			stAxis[GVL.cXM].mcMoveAbs(Axis:=stAxis[GVL.cXM].axisRef, Position:=GVL.cPosEnd, Velocity:=fSpeed, Acceleration:=fAccel, Deceleration:=fAccel, Jerk:=fJerk, Execute:=TRUE);
		END_IF
		
		IF nExt = GVL.cXP THEN
			stAxis[GVL.cXP].mcMoveAbs(Axis:=stAxis[GVL.cXP].axisRef, Position:=GVL.cPosEnd, Velocity:=fSpeed, Acceleration:=fAccel, Deceleration:=fAccel, Jerk:=fJerk, Execute:=TRUE);
		ELSIF nExt = GVL.cXM THEN	
			stAxis[GVL.cXM].mcMoveAbs(Axis:=stAxis[GVL.cXM].axisRef, Position:=GVL.cPosStart, Velocity:=fSpeed, Acceleration:=fAccel, Deceleration:=fAccel, Jerk:=fJerk, Execute:=TRUE);
		END_IF
	
		IF stAxis[GVL.cXP].mcMoveAbs.Done THEN
			stAxis[GVL.cXP].mcMoveAbs(Axis:=stAxis[GVL.cXP].axisRef, Execute:=FALSE);
			nNextState := 1410;
		END_IF			
		IF stAxis[GVL.cXM].mcMoveAbs.Done THEN
			stAxis[GVL.cXM].mcMoveAbs(Axis:=stAxis[GVL.cXM].axisRef, Execute:=FALSE);
			nNextState := 1410;
		END_IF	
		
	1410: //End action
		bBusy := FALSE;

END_CASE

END_FUNCTION_BLOCK

// ---- POUs/StateMachine/StateTop/StateEnabled/FB_Reset.TcPOU
FUNCTION_BLOCK FB_Reset
VAR_IN_OUT
	stAxis 	 	: ARRAY [GVL.cXP .. GVL.cXM] OF ST_AxisGroup;	
	bResetting	: BOOL;
	bResetEntry : BOOL;
END_VAR
VAR
	nCurrentState 	: INT;
	nNextState		: INT := 100;
	//a,b,c,d,e : INT;
	fbResetTimer	: TON ;
END_VAR

IF bResetEntry THEN
	nNextState := 50;
	bResetEntry := FALSE;
END_IF

nCurrentState := nNextState;
CASE nCurrentstate OF
	
	50:
		stAxis[GVL.cXP].mcReset(axis:=stAxis[GVL.cXP].axisRef, Execute:=TRUE);
		stAxis[GVL.cXM].mcReset(axis:=stAxis[GVL.cXM].axisRef, Execute:=TRUE);
		IF stAxis[GVL.cXP].mcReset.Done AND stAxis[GVL.cXM].mcReset.Done THEN
			stAxis[GVL.cXP].mcReset(axis:=stAxis[GVL.cXP].axisRef, Execute:=FALSE);
			stAxis[GVL.cXM].mcReset(axis:=stAxis[GVL.cXM].axisRef, Execute:=FALSE);
			nNextState := 100;
		END_IF
		//e := e+1;
		
	100:
		stAxis[GVL.cXP].mcStop(Axis:=stAxis[GVL.cXP].axisRef, Execute:=FALSE);
		stAxis[GVL.cXM].mcStop(Axis:=stAxis[GVL.cXM].axisRef, Execute:=FALSE);
		fbResetTimer(IN:=TRUE, PT:=T#100MS);
		IF FBResetTimer.Q THEN
			fbResetTimer(IN:=FALSE);
			nNextState:=200;
		END_IF
		//nNextState := 200;
		//a := a+1;
		
	200:
		stAxis[GVL.cXP].mcStop(Axis:=stAxis[GVL.cXP].axisRef, Execute:=TRUE);
		stAxis[GVL.cXM].mcStop(Axis:=stAxis[GVL.cXM].axisRef, Execute:=TRUE);
		IF stAxis[GVL.cXP].mcStop.Done AND stAxis[GVL.cXM].mcStop.Done THEN 
			stAxis[GVL.cXP].mcStop(Axis:=stAxis[GVL.cXP].axisRef, Execute:=FALSE);
			stAxis[GVL.cXM].mcStop(Axis:=stAxis[GVL.cXM].axisRef, Execute:=FALSE);
			nNextState := 300;
			//b := b+1;
		END_IF
		//c := c+1;
	
